// ---- POUs/_Exclude/FB_PACK_WriteOCVFileLoop_v3.TcPOU
(* scan and validate Outers, generate OAC file for new valid Outers *)
FUNCTION_BLOCK FB_PACK_WriteOCVFileLoop_v3
VAR_INPUT
	bExecute						: BOOL;			(* scan for completed Outer *)
	ePackAggregationMode			: E_SYSTEM_PackAggregationMode ;
	strLocalOCVPath				: STRING(50);	(* OCV folder path *)
	nPacksPerOuter				: INT;
	nPackPos1						: INT 	:=1;
	nPackPos2						: INT	:=2;
	nOCVControlCheckStatus		: BYTE;
	aDisablePackAggregCamera	: ARRAY[1..3] OF BOOL;
	stDuplicatedItem				: ST_RejectItems;(*stPackRejectReasons.stPackCodesDuplicated*)
	stCTDateTime					: ST_SYSTEM_DateTime;
END_VAR
VAR_IN_OUT
	stCodeInfo_Pack				: ST_CodeInfo;
	stCodeInfo_Intermediate		: ST_CodeInfo;
	(*aInterimCodeQueue			: ARRAY[1..cMAX_INTERMEDIATE_CODE_QUEUE] OF T_MaxString;*)
	aOCVPackStatus				: ARRAY[1..cMAX_OUTER_STATUS_QUEUE] OF ST_OUTER_Status;	(* Outer status array *)
	stMetsEfficiency				: ST_NOVRAM_METS_Inspection;
	stShiftItemProduced			: ST_KPI_ItemsProduced;
	stProdItemProduced			: ST_KPI_ItemsProduced;
	stLastOCVStatus				: ST_OUTER_Status;	(* Outer status *)
END_VAR
VAR_OUTPUT
	bDone							: BOOL;			(* TRUE = validation complete *)
	bBusy							: BOOL;			(* TRUE = validation in progress *)
	bError							: BOOL;			(* TRUE = validation error *)
	nErrorID						: UDINT;			(* error ID *)
	sOCVFile1						: T_OCV_Filename;	(* OCV file name *)
	sOCVFile2						: T_OCV_Filename;	(* OCV file name *)
	sDeletedOCVFile1				: T_OCV_Filename;
	sDeletedOCVFile2				: T_OCV_Filename;
	bPackCodeDuplicate			: BOOL;
	bInterimCodeDuplicate		: BOOL;
	nWriteOCVError				: UINT;
	nLastTriggerID					: UDINT;
	nOCVFilesCreated				: UDINT;			(* OCV files created *)
	nOCVFilesDeleted				: UINT;
	nOutersStoredInOCV			: UDINT;
	nLinkedPackInOCV				: UDINT;
	nWriteErrorCounter			: UINT;
	bOCVUpdated					: BOOL;
	bOCVValidated					: BOOL;
	stLastValidatedOCV			: ST_OUTER_Status;	(* Outer status *)
	sPackCodesResultToOCV		: T_LongSTRING;
END_VAR
VAR
	fbExecute					: R_TRIG;
	tonTimeOut				: TON;
	rtTimeOutExec				: R_TRIG;
	eState						: E_OCV_State;
	eErrorState					: E_OCV_State;
	eCodeAIType				: E_CodeAIType;
	nMaxOuterIndex			: INT;
	nOuterIndex				: INT;
	nSourceIndex				: INT;
	nPackIndex				: INT;

	bUseIntermediateCode		: BOOL;
	stOCVStatus				: ST_OUTER_Status;	(* Outer status *)

(******************************************************************************)

	fbChekcDupPackCode			: FB_PACK_DuplicatesPackCodes;
	fbPackInspectionEfficency		: FB_KPI_PackEfficiency;
	fbValidateOCVContent			: FB_PACK_ValidateOCVContent;

	aAggregationCodesValid			: ARRAY[1..2] OF  BOOL;
	aDeleteOCVCodesValid			: ARRAY[1..2] OF BOOL;
(******************************************************************************)

	fbWriteOCVFile				: FB_OCV_WriteFile;
	(*sOCVFileName				: T_MaxString;*)
	fbMoveOCVFile			: FB_FILE_Move;

	nOCVLogIndex		: UINT;
	sLocalTargetPath	: STRING(255);

END_VAR


(* monitor rising edge of bExecute *)
fbExecute(CLK := bExecute);

(* monitor Busy timeout *)
tonTimeOut(
	IN:=nSourceIndex <> 0,
	 PT:=cONE_SECOND,
	Q=>
);

rtTimeOutExec(CLK:= tonTimeOut.Q);

IF rtTimeOutExec.Q THEN

	bError := TRUE;
	nErrorID := 100;
	IF nSourceIndex > 0 THEN

		aOCVPackStatus[nSourceIndex].sDataSourceTracker 	:= 	'TIMEOUT_S';
		aOCVPackStatus[nSourceIndex].nStatus.7 := TRUE;

		stLastOCVStatus := aOCVPackStatus[nSourceIndex];
		bOCVUpdated	:= TRUE;
		stLastValidatedOCV := aOCVPackStatus[nSourceIndex];
		bOCVValidated	:= TRUE;
	END_IF

	eState := E_OCV_DONE;
END_IF

(* rising edge of bExecute *)
CASE eState OF

	(* idle *)
	E_OCV_IDLE:

		(* scan for completed Outer when OAC files are required *)
		IF fbExecute.Q = TRUE THEN

			(* update outputs *)
			bDone := FALSE;
			bBusy := TRUE;
			bError := FALSE;
			nErrorID := 0;

			(* clear outputs *)
			nOCVFilesCreated := 0;
			nOutersStoredInOCV := 0;
			nLinkedPackInOCV :=0;
			nWriteErrorCounter :=0;

			(*bOCVUpdated	:= FALSE;*)

			(* max Outer index *)
			nMaxOuterIndex := UDINT_TO_INT(SIZEOF(aOCVPackStatus) / SIZEOF(aOCVPackStatus[1]));

			eState := E_OCV_SCAN;

		(* no action required *)
		ELSIF bExecute = FALSE THEN

			(* reset outputs *)
			bDone := FALSE;
			bBusy := FALSE;
			bError := FALSE;
			nErrorID := 0;

		END_IF

	(* scan for completed Outer *)
	E_OCV_SCAN:

		eState := E_OCV_DONE;
		bOCVUpdated	:= FALSE;
		bOCVValidated	:= FALSE;

		(* reset index of Outer to be written to OCV file *)
		nSourceIndex := 0;
		MEMSET(ADR(aAggregationCodesValid), 16#00, SIZEOF(aAggregationCodesValid));
		MEMSET(ADR(aDeleteOCVCodesValid), 16#00, SIZEOF(aDeleteOCVCodesValid));

		bPackCodeDuplicate			:= FALSE;

		 (* scan aOCVPackStatus  backward - ensures that oldest Outer will be written first *)
		FOR nOuterIndex := nMaxOuterIndex TO 1 BY -1 DO
			CASE ePackAggregationMode OF

			E_SYSTEM_PAOL_3CAM:
				(* TriggerID > 0 indicates Outer data present, nStatus = 14 indicates writing data for all 3 cameras, nStatus.6  indicates OCV file has been alread  created, nStatus.7 indicates OCV write error  *)
				IF aOCVPackStatus[nOuterIndex].nTriggerID > 0 AND
					(aOCVPackStatus[nOuterIndex].nStatus.1 OR aDisablePackAggregCamera[1])	AND
					( aOCVPackStatus[nOuterIndex].nStatus.2 OR aDisablePackAggregCamera[2]) 	AND
					( aOCVPackStatus[nOuterIndex].nStatus.3 OR aDisablePackAggregCamera[3]) 	AND
					NOT aOCVPackStatus[nOuterIndex].nStatus.6 		AND
					NOT aOCVPackStatus[nOuterIndex].nStatus.7  		AND
					NOT aOCVPackStatus[nOuterIndex].nStatus.22		AND
					NOT aOCVPackStatus[nOuterIndex].nStatus.23 	THEN

					(* For lightbox system,mapping packcodes to AggregationCodes, used for file name has to be done here, when we are sure if all pack data was plced to OCV record. Those codes will be used to restore OCV data to OAC*)
					AggregationCodes();

					bUseIntermediateCode := FALSE;
					nSourceIndex := nOuterIndex;
					EXIT;
				END_IF

			E_SYSTEM_PAOL_2CAM:
				(* TriggerID > 0 indicates Outer data present, nStatus = 14 indicates writing data for all 3 cameras, nStatus.6  indicates OCV file has been alread  created, nStatus.7 indicates OCV write error  *)
				IF aOCVPackStatus[nOuterIndex].nTriggerID > 0 AND
					(aOCVPackStatus[nOuterIndex].nStatus.1 OR aDisablePackAggregCamera[1])		AND
					( aOCVPackStatus[nOuterIndex].nStatus.2 OR aDisablePackAggregCamera[2]) 	AND
					NOT aOCVPackStatus[nOuterIndex].nStatus.6 		AND
					NOT aOCVPackStatus[nOuterIndex].nStatus.7  		AND
					NOT aOCVPackStatus[nOuterIndex].nStatus.22		AND
					NOT aOCVPackStatus[nOuterIndex].nStatus.23 	THEN

					(* For lightbox system,mapping packcodes to AggregationCodes, used for file name has to be done here, when we are sure if all pack data was plced to OCV record. Those codes will be used to restore OCV data to OAC*)
					AggregationCodes();

					bUseIntermediateCode := FALSE;
					nSourceIndex := nOuterIndex;
					EXIT;
				END_IF

			E_SYSTEM_PLAS_T01:
				(* TriggerID > 0 indicates Outer data present, nStatus = 14 indicates writing data for all 3 cameras, nStatus.6  indicates OCV file has been alread  created, nStatus.7 indicates OCV write error  *)
				(* For linear aggregation system,AggregationCode shuld be already add from temporary coding system camera. This code will be used for file name and to restore OCV data to OAC*)

				IF aOCVPackStatus[nOuterIndex].nTriggerID > 0 		AND
					aOCVPackStatus[nOuterIndex].nStatus.0			AND 	(*OCV Structure rady to store in file *)
					NOT aOCVPackStatus[nOuterIndex].nStatus.6 		AND
					NOT aOCVPackStatus[nOuterIndex].nStatus.7  		AND
					NOT aOCVPackStatus[nOuterIndex].nStatus.22		AND
					NOT aOCVPackStatus[nOuterIndex].nStatus.23 	THEN

					(* For clear wrap system,mapping packcodes to AggregationCodes, used for file name has to be done here, when we are sure if all pack data was plced to OCV record. Those codes will be used to restore OCV data to OAC*)
					(*AggregationCodes();*)

					bUseIntermediateCode := FALSE;
					nSourceIndex := nOuterIndex;
					EXIT;
				END_IF

			E_SYSTEM_PLAS_T02, E_SYSTEM_PLAS_T03, E_SYSTEM_PLAS_T04:
				(* TriggerID > 0 indicates Outer data present, nStatus = 14 indicates writing data for all 3 cameras, nStatus.6  indicates OCV file has been alread  created, nStatus.7 indicates OCV write error  *)
				(* For linear aggregation system,AggregationCode shuld be already add from temporary coding system camera. This code will be used for file name and to restore OCV data to OAC*)

				IF aOCVPackStatus[nOuterIndex].nTriggerID > 0 		AND
					aOCVPackStatus[nOuterIndex].nStatus.0			AND 	(*OCV Structure rady to store in file *)
					NOT aOCVPackStatus[nOuterIndex].nStatus.6 		AND
					NOT aOCVPackStatus[nOuterIndex].nStatus.7  		AND
					NOT aOCVPackStatus[nOuterIndex].nStatus.22		AND
					NOT aOCVPackStatus[nOuterIndex].nStatus.23 	THEN

					(* For NON clear wrap system,mapping packcodes to AggregationCodes form Intrim code, which might be temp stored as barcode for OCV records.
						AggregationCode1 will be used for file name has to be done here, when we are sure if all pack data was plced to OCV record. Those codes will be used to restore OCV data to OAC*)
						(*aOCVPackStatus[nOuterIndex].stOACData.AggregationCodes[1] :=aOCVPackStatus[nOuterIndex].stOACData.Barcode;*) (*solution never tested yet*)

					bUseIntermediateCode := TRUE;
					nSourceIndex := nOuterIndex;
					EXIT;
				END_IF
			END_CASE
		END_FOR

		(* Outer found requiring OAC file to be written *)
		IF nSourceIndex > 0 THEN

			(* copy Outer data from arrOuterStatus *)
			stOCVStatus := aOCVPackStatus[nSourceIndex];

			stMetsEfficiency.OutersProcessing.AtPackAggregCameras := stMetsEfficiency.OutersProcessing.AtPackAggregCameras  + 1;

			eState := E_OCV_VALIDATECONTENT;
		END_IF

	E_OCV_VALIDATECONTENT:

		fbChekcDupPackCode(
			nNumberPackInOuters := nPacksPerOuter,
			sOuterStatus := stOCVStatus,
			stDuplicatedItem := stDuplicatedItem,
			bDuplicateFound =>  bPackCodeDuplicate
			);

		fbPackInspectionEfficency(
			ePackAggregationMode				:= ePackAggregationMode,
			nTotalOutersProcessingByPackAggregCameras	:= stMetsEfficiency.OutersProcessing.AtPackAggregCameras,
			bUseInterimCode						:= bUseIntermediateCode,
			sOuterStatus							:= stOCVStatus,
			aPacksRead							:= stMetsEfficiency.PacksRead,
			aPackPosEfficiency						:= stMetsEfficiency.PackPosEfficiency,
			stPackAggregationEfficiency			:= stMetsEfficiency.PackAggregationEfficiency,
			stMainItemProduced					:= stMetsEfficiency.PackProduced,
			stShiftItemProduced					:= stShiftItemProduced,
			stProdItemProduced					:= stProdItemProduced
			);

		fbValidateOCVContent(
			nOCVControlCheckStatus			:= nOCVControlCheckStatus,
			nPacksPerOuter					:= nPacksPerOuter,
			stCTDateTime						:= stCTDateTime,
			bUseIntermediateCode				:= bUseIntermediateCode,
			stCodeInfo_Pack					:= stCodeInfo_Pack,
			stCodeInfo_Intermediate			:= stCodeInfo_Intermediate,
			(*aInterimCodeQueue				:= aInterimCodeQueue,*)
			stOCVStatus						:= stOCVStatus,
			stNextOCVStatus					:= aOCVPackStatus[nSourceIndex+1],
			bDuplicateInterimFound			=> bInterimCodeDuplicate
			);


		stLastValidatedOCV := stOCVStatus; (*Use for logging data*)
		bOCVValidated	:= TRUE;	(*Use for SFLX solution*)

		IF F_InvalidateASCIIChar(fbValidateOCVContent.aOCVFileCodeName[1]) =	0 	THEN aAggregationCodesValid[1] := nPackPos1 <> 0 OR  bUseIntermediateCode;  	END_IF
		IF F_InvalidateASCIIChar(fbValidateOCVContent.aOCVFileCodeName[2]) =	0 	THEN aAggregationCodesValid[2] := nPackPos2 <> 0; 		END_IF

		IF (aAggregationCodesValid[1] OR aAggregationCodesValid[2]) THEN
			eState := E_OCV_WRITEDATA;
		ELSE

			stOCVStatus.nStatus.7 := TRUE;

			IF fbValidateOCVContent.bDuplicatePackFound THEN
				eState := E_OCV_MOVEFILE1;
			ELSE
				eState := E_OCV_UPDATESTATUS;
			END_IF

			nWriteErrorCounter := nWriteErrorCounter+1;
		END_IF

	(* write OCVC file *)
	E_OCV_WRITEDATA:

		IF fbValidateOCVContent.bEmptyAggregationCode 		THEN

			sLocalTargetPath := CONCAT(strLocalOCVPath,'Empty\');

		ELSIF fbValidateOCVContent.bInvalidPackFound 			OR
				fbValidateOCVContent.bDuplicatePackFound 		OR
				fbValidateOCVContent.bDuplicateInterimFound 	THEN

			sLocalTargetPath := CONCAT(strLocalOCVPath,'Error\');
		ELSE
			sLocalTargetPath := strLocalOCVPath;
		END_IF

		(* write OCV file *)
		fbWriteOCVFile(
			bExecute					:= TRUE,
			sTargetPath				:= sLocalTargetPath,
			ePackAggregationMode	:= ePackAggregationMode,
			nPacksPerOuter			:= nPacksPerOuter,
			aOCVFileCodeName		:= fbValidateOCVContent.aOCVFileCodeName,  (*strAggregationCodes is a table*)
			bSkipWriteFile1			:= NOT aAggregationCodesValid[1],
			bSkipWriteFile2			:= NOT aAggregationCodesValid[2],
			stOCVPackStatus			:= stOCVStatus
			);
		(* write OCV file complete *)
		IF fbWriteOCVFile.bDone  THEN

			sOCVFile1 := fbWriteOCVFile.sOCVFile1;
			sOCVFile2 := fbWriteOCVFile.sOCVFile2;

			(* write OCV file completed OK *)
			IF NOT  fbWriteOCVFile.bError THEN

				(* count OCV files written *)
				nOCVFilesCreated := nOCVFilesCreated + fbWriteOCVFile.nStoredFiles;
				nOutersStoredInOCV := nOutersStoredInOCV + 1;

				nLastTriggerID :=  stOCVStatus.nTriggerID;

				(* update stOCVStatus - OCV file written OK *)
				stOCVStatus.nStatus.6 := TRUE;
			ELSE
				bError := TRUE;
				nErrorID := fbWriteOCVFile.nErrorID + 1000;

				(* update stOCVStatus - OCV file write error  - general error for OCV *)
				nWriteOCVerror := nWriteOCVerror +1;
				stOCVStatus.nStatus.7 := TRUE;
				eErrorState := eState;
			END_IF

			IF fbValidateOCVContent.bDuplicatePackFound  THEN
				eState := E_OCV_MOVEFILE1;
			ELSE
				eState := E_OCV_UPDATESTATUS;
			END_IF
			(* close off fbWriteOCVFile*)
			fbWriteOCVFile(bExecute := FALSE);
		END_IF

	(* delete OCV to error folder *)
	E_OCV_MOVEFILE1:

		IF F_InvalidateASCIIChar(fbValidateOCVContent.aOCVFileCodeToDelete[1]) = 0 	THEN aDeleteOCVCodesValid[1] := nPackPos1 <> 0 OR  bUseIntermediateCode;  	END_IF

		(*sOCVFileName := F_CONCAT3('OCV_', fbValidateOCVContent.aOCVFileCodeToDelete[1], '.xml');*)
		(* delete OCV file *)
		fbMoveOCVFile(
				bExecute			:= aDeleteOCVCodesValid[1],
				strPathSource		:= strLocalOCVPath,
				strPathTarget		:= CONCAT(strLocalOCVPath,'Error\' ),
				strFileName		:= fbValidateOCVContent.aOCVFileCodeToDelete[1],
				tTimeout			:= cHALF_SECOND
		);

		(* delete file complete *)
		IF NOT fbMoveOCVFile.bBusy  OR NOT aDeleteOCVCodesValid[1] THEN

			(* delete  file completed OK *)
			IF NOT  fbMoveOCVFile.bError THEN

				(* update counter *)
				IF  aDeleteOCVCodesValid[1] THEN
					nOCVFilesDeleted := nOCVFilesDeleted + 1;
					sDeletedOCVFile1 := fbMoveOCVFile.strLastFileMoved;
				END_IF
			(* delete command error or file not found *)
			ELSE

				bError := TRUE;
				nErrorID := fbMoveOCVFile.nErrorID + 2000;
				eErrorState := eState;
			END_IF

			(* close off fbDeleteOCVFile *)
			fbMoveOCVFile(bExecute := FALSE);

			eState := E_OCV_MOVEFILE2;
		END_IF

	(* delete OCV to error folder *)
	E_OCV_MOVEFILE2:

		IF F_InvalidateASCIIChar(fbValidateOCVContent.aOCVFileCodeToDelete[2]) = 0 	THEN aDeleteOCVCodesValid[2] := nPackPos2 <> 0; 		END_IF

		(*sOCVFileName := F_CONCAT3('OCV_', fbValidateOCVContent.aOCVFileCodeToDelete[2], '.xml');*)
		(* delete OCV file *)
		fbMoveOCVFile(
				bExecute			:= aDeleteOCVCodesValid[2],
				strPathSource		:= strLocalOCVPath,
				strPathTarget		:= CONCAT(strLocalOCVPath,'Error\' ),
				strFileName		:= fbValidateOCVContent.aOCVFileCodeToDelete[2],
				tTimeout			:= cHALF_SECOND
		);

		(* delete file complete *)
		IF NOT fbMoveOCVFile.bBusy  OR NOT aDeleteOCVCodesValid[2] THEN

			(* delete  file completed OK *)
			IF NOT  fbMoveOCVFile.bError  THEN

				(* update counter *)
				IF aDeleteOCVCodesValid[2] THEN
					nOCVFilesDeleted := nOCVFilesDeleted + 1;
					sDeletedOCVFile2 := fbMoveOCVFile.strLastFileMoved;
				END_IF
			(* delete command error or file not found *)
			ELSE

				bError := TRUE;
				nErrorID := fbMoveOCVFile.nErrorID + 3000;
				eErrorState := eState;
			END_IF
			(* close off fbDeleteOCVFile *)
			fbMoveOCVFile(bExecute := FALSE);

			eState := E_OCV_UPDATESTATUS;
		END_IF

	(* update Outer status *)
	E_OCV_UPDATESTATUS:

		nSourceIndex := 0;
		(* move stOCVStatus data back to shift reg *)
		FOR nOuterIndex := 1 TO nMaxOuterIndex DO

			(* matching nTriggerID found *)
			IF aOCVPackStatus[nOuterIndex].nTriggerID = stOCVStatus.nTriggerID THEN

				(* move updated Outer data to shift reg *)
				aOCVPackStatus[nOuterIndex] := stOCVStatus;
				stLastOCVStatus := stOCVStatus;

				nLinkedPackInOCV :=nLinkedPackInOCV + stOCVStatus.stOACData.NumberOfLinkedPacks;
				bOCVUpdated	:= TRUE;

				sPackCodesResultToOCV	:= '';
				sPackCodesResultToOCV := F_CONCAT5('[', RIGHT(stLastOCVStatus.stOACData.AggregationCodes[1],7),']:[',RIGHT(stLastOCVStatus.stOACData.AggregationCodes[2],7),']');
				FOR nOCVLogIndex := 1 TO MIN(nPacksPerOuter ,cMAX_PACKS_PER_OUTER) BY 1 DO
					sPackCodesResultToOCV :=F_LongCONCAT(sPackCodesResultToOCV, '     ');
					sPackCodesResultToOCV := F_LongCONCAT(sPackCodesResultToOCV, RIGHT(F_CODE_GetItem(stLastOCVStatus.stOACData.PackCode[nOCVLogIndex], eCodeAIType.SerialCode, stCodeInfo_Pack),7));
				END_FOR

				EXIT;
			END_IF
		END_FOR

		eState := E_OCV_SCAN;

	(* OCV file complete *)
	E_OCV_DONE:

		(* update outputs *)
		bDone := TRUE;
		bBusy := FALSE;

		eState := E_OCV_IDLE;

(* unknown state *)
ELSE

	eState := E_OCV_IDLE;
END_CASE

ACTION AggregationCodes:
IF nPackPos1 <> 0 THEN
	IF aOCVPackStatus[nOuterIndex].aOACPackStatus[nPackPos1] > 1 THEN
		aOCVPackStatus[nOuterIndex].stOACData.AggregationCodes[1] :=aOCVPackStatus[nOuterIndex].stOACData.PackCode[nPackPos1];
	ELSE
		aOCVPackStatus[nOuterIndex].stOACData.AggregationCodes[1] := '';
	END_IF
ELSE
	aOCVPackStatus[nOuterIndex].stOACData.AggregationCodes[1] := '';
END_IF

IF nPackPos2 <> 0 THEN
	IF aOCVPackStatus[nOuterIndex].aOACPackStatus[nPackPos2] > 1 THEN
		aOCVPackStatus[nOuterIndex].stOACData.AggregationCodes[2] :=aOCVPackStatus[nOuterIndex].stOACData.PackCode[nPackPos2];
	ELSE
		aOCVPackStatus[nOuterIndex].stOACData.AggregationCodes[2] := '';
	END_IF
ELSE
	aOCVPackStatus[nOuterIndex].stOACData.AggregationCodes[2] := '';
END_IF
END_ACTION

END_FUNCTION_BLOCK

// ---- POUs/_Exclude/FB_T03_MoveDataToOCVStatus_ORG.TcPOU
FUNCTION_BLOCK FB_T03_MoveDataToOCVStatus_ORG
VAR_INPUT
	bExecute						: BOOL;

	stImageData					: ST_SCANNER_ImageData;	(* image data structure *)
	nExpectedResp					: INT:=1;
	(*nExpectedValidationDepth		: INT;*)
	nPacksPerOuter				: UINT;
	bConfirmOnOuter				: BOOL;
END_VAR
VAR_IN_OUT
	stPackRejectReasons			: ST_RejectReasonsForPack;
	stPackInFeedQueue			: ST_PACK_InfeedQueue; (* Infeed queue *)
	stOCVPackStatus				: ST_OUTER_Status;
	stCodeInfo						: ST_CodeInfo;
END_VAR
VAR_OUTPUT
	bDone							: BOOL;

	nImageDataIndex				: UINT;
	nSearchIndex					: UINT;
	nMoveIndex					: UINT;
	nValidatinIndex				: UINT;

	bOCVStackOutOfSequence		: BOOL;
	bOCVNoConfiramtion			: BOOL;
	bOCVConfirmationNotFound	: BOOL;

	sStackerDataLog				: T_LongSTRING;
END_VAR
VAR
	fbExecute						: R_TRIG;

	nPackIndex					: UINT;
	nLogIndex						: INT;

	nValidationOffset 				: INT;

	aDiagonosticError				: ARRAY[1..10] OF INT;
	aDiagonosticMove				: ARRAY[0..20] OF INT;
END_VAR

VAR CONSTANT
	aPackCodeMapping2x5		: ARRAY[1..cMAX_PACKS_PER_OUTER] OF INT :=[ 	9, 8, 7, 6, 5, 4, 3, 2, 1, 0];		(*mapping examples*)
	aPackCodeMapping5x2		: ARRAY[1..cMAX_PACKS_PER_OUTER] OF INT :=[ 	0, 1, 2, 3, 4, 5, 6, 7, 8, 9];		(*mapping examples*)
END_VAR

fbExecute(CLK := bExecute);

IF fbExecute.Q THEN

	bDone := FALSE;
	nMoveIndex	:= 0;
	nSearchIndex 	:=0;		(*initialize in for loop on 1*)
	nImageDataIndex := 0;	(*initialize in for loop on 1*)

	sStackerDataLog	:= '';

	bOCVStackOutOfSequence		:= FALSE;
	bOCVNoConfiramtion			:= FALSE;
	(*bOCVConfirmationNotFound	:= FALSE;*)

	(*nExpectedValidationDepth	:= LIMIT(1, nExpectedValidationDepth, cMAX_CAMERA_PROG_NUMBER);*)

	nValidationOffset :=SEL(bConfirmOnOuter, 0, nExpectedResp);

(*********************************Identify index***************************************************)

	IF stImageData.nCodesRead > 0 THEN

		FOR nImageDataIndex := 1 TO stImageData.nCodesRead DO
			FOR nSearchIndex :=1 TO cMAX_PACK_INFEED_QUEUE DO

				IF stImageData.aCodeData[nImageDataIndex].strDataString  = stPackInFeedQueue.aPackQueue[nSearchIndex].sPackCode AND
					stPackInFeedQueue.aPackQueue[nSearchIndex].sPackCode <> '' THEN

					IF nSearchIndex > stImageData.aCodeData[nImageDataIndex].nProgramNo THEN
						nMoveIndex := nSearchIndex-stImageData.aCodeData[nImageDataIndex].nProgramNo +nValidationOffset;  (*add nExpectedResp as an option*)
						EXIT;
					END_IF
				END_IF
			END_FOR

			IF nMoveIndex > 0 THEN
				EXIT;
			END_IF
		END_FOR

	ELSIF stImageData.nCodesRead = 0 AND stPackInFeedQueue.nIndex = nPacksPerOuter THEN
		
		nMoveIndex := stPackInFeedQueue.nIndex;
	END_IF

sStackerDataLog	:= F_CONCAT3('MOVED ITEM [', UINT_TO_STRING(nMoveIndex), ']:');

(*********************************Validation***************************************************)

	IF	bOCVConfirmationNotFound AND nMoveIndex <> 0 THEN		(*reject next outer after one with read code bou confirmation not found*)

		sStackerDataLog	:= CONCAT(sStackerDataLog, '[X]');

		aDiagonosticError[1]	:=  aDiagonosticError[1] + 1;
		bOCVConfirmationNotFound := FALSE;
		bOCVStackOutOfSequence := TRUE;

	ELSIF	stImageData.nCodesRead = 0 AND nMoveIndex = nPacksPerOuter THEN		(*move without confirmation found - temp blocked*)

		aDiagonosticError[2]	:=  aDiagonosticError[2] + 1;
		bOCVNoConfiramtion := TRUE;

	ELSIF nMoveIndex = 0 AND stImageData.nCodesRead <> 0 THEN			(*Confirmation code read but not found in infeed*)

		sStackerDataLog	:= CONCAT(sStackerDataLog, '[Y]');

		aDiagonosticError[3]	:=  aDiagonosticError[3] + 1;
		bOCVConfirmationNotFound := TRUE;

	ELSIF nMoveIndex = 0 THEN		(*Confirmation code not found becouse camera not read*)

		sStackerDataLog	:= CONCAT(sStackerDataLog, '[Z]');

		aDiagonosticError[4]	:=  aDiagonosticError[4] + 1;
		bOCVConfirmationNotFound := TRUE;

	ELSIF  stImageData.nCodesRead <> nExpectedResp (*nExpectedValidationDepth*) THEN	(*no read or not enough code read found but at leas one code read and found*)

		aDiagonosticError[5]	:=  aDiagonosticError[5] + 1;
		bOCVStackOutOfSequence := TRUE;

	ELSIF nMoveIndex > nPacksPerOuter THEN		(*f.ex phisical packs remode form line*)

		aDiagonosticError[6]	:=  aDiagonosticError[6] + 1;
		bOCVStackOutOfSequence := TRUE;

	ELSIF nMoveIndex < nPacksPerOuter THEN		(*f.ex phantom packs passed form the line or queue was deleted*)

		aDiagonosticError[7]	:=  aDiagonosticError[7] + 1;
		bOCVStackOutOfSequence := TRUE;

		IF nMoveIndex < 20 THEN	aDiagonosticMove[nMoveIndex] :=  aDiagonosticMove[nMoveIndex] + 1; END_IF

		aDiagonosticError[8]	:=  aDiagonosticError[8] + 1;
		bOCVStackOutOfSequence := TRUE;

	ELSIF nMoveIndex = nPacksPerOuter  AND
			stImageData.nCodesRead > 0	AND
			nMoveIndex  <= cMAX_PACK_INFEED_QUEUE - cMAX_CAMERA_PROG_NUMBER	THEN

		(*Check all reaming codes in the comfirmation stack*)
		FOR nValidatinIndex := 1 TO stImageData.nCodesRead DO														(*nMovePsotion - nExpectedResp as an option*)
			IF stImageData.aCodeData[nValidatinIndex].strDataString <> stPackInFeedQueue.aPackQueue[nMoveIndex + stImageData.aCodeData[nValidatinIndex].nProgramNo - nValidationOffset].sPackCode(* AND
				stPackInFeedQueue.aPackQueue[nMoveIndex + stImageData.aCodeData[nValidatinIndex].nProgramNo - nValidationOffset].sPackCode <> ''*)  THEN (*More restricted to reject if comapre with empty*)

				aDiagonosticError[9]	:=  aDiagonosticError[9] + 1;
				bOCVStackOutOfSequence := TRUE;
				EXIT;
			END_IF
		END_FOR
	ELSE
		aDiagonosticError[10]	:=  aDiagonosticError[10] + 1;
		bOCVStackOutOfSequence := TRUE;
	END_IF

(*********************************Fill up OCV pack data***************************************************)

	IF NOT bOCVStackOutOfSequence 		AND
		NOT bOCVNoConfiramtion 			AND
		NOT bOCVConfirmationNotFound  	THEN		(*temp for now included bOCVNoConfiramtion*)

		FOR nPackIndex := 1 TO LIMIT(1, nPacksPerOuter, cMAX_PACKS_PER_OUTER) DO

			(* to avoid incorect mapping in PackCodeMapping declaration, where array index <0 *)
			IF nMoveIndex >  aPackCodeMapping2x5[nPackIndex] AND nPacksPerOuter > 0 THEN
				stOCVPackStatus.stOACData.PackCode[nPackIndex] := stPackInFeedQueue.aPackQueue[nMoveIndex - aPackCodeMapping2x5[nPackIndex]].sPackCode;
				stOCVPackStatus.aPackCodeFilledIn[nPackIndex] := stPackInFeedQueue.aPackQueue[nMoveIndex -aPackCodeMapping2x5[nPackIndex]].ePackCodeFilledIn;
				stOCVPackStatus.aPackCodes[nPackIndex].sBuffer[1].strCode := stPackInFeedQueue.aPackQueue[nMoveIndex -aPackCodeMapping2x5[nPackIndex]].stPackCodeData.strDataString;

				stOCVPackStatus.aOACPackStatus[nPackIndex]	:= stPackInFeedQueue.aPackQueue[nMoveIndex -aPackCodeMapping2x5[nPackIndex]].nPackStatus;
				stOCVPackStatus.stOACData.PackRejectID[nPackIndex] :=  stPackInFeedQueue.aPackQueue[nMoveIndex -aPackCodeMapping2x5[nPackIndex]].nPackRejectID;
				stOCVPackStatus.stOACData.PackRejectCode[nPackIndex] := stPackInFeedQueue.aPackQueue[nMoveIndex -aPackCodeMapping2x5[nPackIndex]].sPackRejectCode;
			ELSE
				EXIT;  	(*stOCVPackStatus remain empty - wrong input parameters*)
			END_IF
		END_FOR
	ELSE

		FOR nPackIndex := 1 TO LIMIT(1, nPacksPerOuter, cMAX_PACKS_PER_OUTER) DO

			IF nPacksPerOuter > 0 THEN
				stOCVPackStatus.stOACData.PackCode[nPackIndex] :=  cCODE_OVERWIRTTEN;
				stOCVPackStatus.aPackCodeFilledIn[nPackIndex] := E_PACK_CODEOVERWRITTEN;
				stOCVPackStatus.aPackCodes[nPackIndex].sBuffer[1].strCode :=  cCODE_OVERWIRTTEN;
		
				stOCVPackStatus.aOACPackStatus[nPackIndex]	:= 1;
				stOCVPackStatus.stOACData.PackRejectID[nPackIndex] :=  stPackRejectReasons.stPackCodesOverwritten.nRejectID;
				stOCVPackStatus.stOACData.PackRejectCode[nPackIndex] := stPackRejectReasons.stPackCodesOverwritten.sMetsDisplayCode;
			ELSE
				EXIT;	(*stOCVPackStatus remain empty - wrong input parameters*)
			END_IF
		END_FOR
	END_IF

(*********************************Log Move Pack Infeed Queue***************************************************)

	IF nMoveIndex <> 0 THEN
		FOR nLogIndex :=1 TO nMoveIndex  DO
			sStackerDataLog :=F_LongCONCAT(sStackerDataLog, '   ');
			sStackerDataLog :=F_LongCONCAT(sStackerDataLog, RIGHT(F_CODE_GetItem(stPackInFeedQueue.aPackQueue[nLogIndex].sPackCode, eCodeAIType.SerialCode, stCodeInfo), 5));
		END_FOR
	END_IF

(*********************************Move Pack Infeed Queue***************************************************)

	IF nMoveIndex <> 0 THEN
		(* move remaining Outers forward in sInfeedQueue and update index pointer *)
		IF cMAX_PACK_INFEED_QUEUE  > nMoveIndex  THEN
	
			MEMMOVE(ADR(stPackInFeedQueue.aPackQueue[1]), ADR(stPackInFeedQueue.aPackQueue[nMoveIndex + 1]),
											 (cMAX_PACK_INFEED_QUEUE- nMoveIndex) * SIZEOF(stPackInFeedQueue.aPackQueue[1]));
			stPackInFeedQueue.nIndex := LIMIT(0, stPackInFeedQueue.nIndex - nMoveIndex,cMAX_PACK_INFEED_QUEUE);
	
		END_IF
	
		(* clear all data for empty Packs in PackInFeedQueue -> from Index + 1 till end of queue *)
		IF cMAX_PACK_INFEED_QUEUE > stPackInFeedQueue.nIndex  THEN

			MEMSET(ADR(stPackInFeedQueue.aPackQueue[stPackInFeedQueue.nIndex + 1]), 16#00,
											(cMAX_PACK_INFEED_QUEUE - stPackInFeedQueue.nIndex ) * SIZEOF(stPackInFeedQueue.aPackQueue[1]));
		END_IF
	END_IF
(****************************************************************************************************************************************************************)

	bDone := TRUE;
ELSE
	bDone := FALSE;

END_IF

END_FUNCTION_BLOCK

// ---- POUs/_Exclude/FSS2/FB_FSS2_BuildXMLData.TcPOU
FUNCTION_BLOCK FB_FSS2_BuildXMLData
VAR_INPUT
	bExecute		: BOOL;
	nCartonsPerMasterCase	:UINT	:=50;
END_VAR
VAR_IN_OUT
	stAgregationData	 			: ST_CHM_Data;		(* case data to be written to XML *)
END_VAR
VAR_OUTPUT
	bDone			: BOOL;
	nImageByte		: INT;		(* total bytes for OAC template *)
	arrXMLImage		: ARRAY[0..4096] OF BYTE;
END_VAR
VAR
	fbExecute		: R_TRIG;
	nOuterIndex		: INT;		(* Outer index when building for CAC file *)

	strString		: STRING(255);
	(*nStringLen		: INT;*)

END_VAR

(* rising edge of bExecute *)
fbExecute(CLK := bExecute);

(* rising edge of bExecute *)
IF fbExecute.Q = TRUE THEN

	(* update outputs *)
	bDone := FALSE;

	(* clear output array and reset byte counter *)
	MEMSET(ADR(arrXMLImage), 16#00, SIZEOF(arrXMLImage));
	nImageByte := 0;


(********************XML FILE BIULD SEQTION****************************)
(* XML file version *)
strString := '<?xml version="1.0" encoding="utf-8"?>$R$N';
MEMMOVE(ADR(arrXMLImage[nImageByte]), ADR(strString), LEN(strString));
nImageByte := nImageByte + LEN(strString);

(* XPath leading tag *)
strString := '<GenericHierarchyList xmlns:xsi="http://www.w3.org/2001/XMLSchema-instance" xsi:noNamespaceSchemaLocation="TNTGenericHierarchy.xsd"> $R$N';
MEMMOVE(ADR(arrXMLImage[nImageByte]), ADR(strString), LEN(strString));
nImageByte := nImageByte + LEN(strString);

	(* RequestID *)
	strString := F_CONCAT3('$T<RequestID>','' , '</RequestID>$R$N');
	MEMMOVE(ADR(arrXMLImage[nImageByte]), ADR(strString), LEN(strString));
	nImageByte := nImageByte + LEN(strString);

	(* Sender *)
	strString := F_CONCAT3('$T<Sender>', 'TNTLS' , '</Sender>$R$N');
	MEMMOVE(ADR(arrXMLImage[nImageByte]), ADR(strString), LEN(strString));
	nImageByte := nImageByte + LEN(strString);

	(* GenericHierarchy *)
	strString := '$T<GenericHierarchy>$R$N';
	MEMMOVE(ADR(arrXMLImage[nImageByte]), ADR(strString), LEN(strString));
	nImageByte := nImageByte + LEN(strString);

		(* User *)
		strString := F_CONCAT3('$T$T<User>','TNTLS', '</User>$R$N');
		MEMMOVE(ADR(arrXMLImage[nImageByte]), ADR(strString), LEN(strString));
		nImageByte := nImageByte + LEN(strString);

		(* Timestamp *)
		strString := F_CONCAT3('$T$T<Timestamp>', stAgregationData.MessageHeader.CreationTimeLocalUTC, '</Timestamp>$R$N');
		MEMMOVE(ADR(arrXMLImage[nImageByte]), ADR(strString), LEN(strString));
		nImageByte := nImageByte + LEN(strString);

		(* PackLevel *)
		strString := F_CONCAT3('$T$T<PackLevel>','MASTERCASE', '</PackLevel>$R$N');
		MEMMOVE(ADR(arrXMLImage[nImageByte]), ADR(strString), LEN(strString));
		nImageByte := nImageByte + LEN(strString);

		(* Parent *)
		strString := '$T$T<Parent>$R$N';
		MEMMOVE(ADR(arrXMLImage[nImageByte]), ADR(strString), LEN(strString));
		nImageByte := nImageByte + LEN(strString);
	
			(* ID *)
			strString := F_CONCAT3('$T$T$T<ID>',stAgregationData.GenericHierarchy.CaseItem.Identity.ID, '</ID>$R$N');
			MEMMOVE(ADR(arrXMLImage[nImageByte]), ADR(strString), LEN(strString));
			nImageByte := nImageByte + LEN(strString);
	
			(* GTIN *)
			strString := F_CONCAT3('$T$T$T<GTIN>', stAgregationData.GenericHierarchy.CaseItem.Identity.GTIN, '</GTIN>$R$N');
			MEMMOVE(ADR(arrXMLImage[nImageByte]), ADR(strString), LEN(strString));
			nImageByte := nImageByte + LEN(strString);

		(*/Parent *)
		strString := '$T$T</Parent>$R$N';
		MEMMOVE(ADR(arrXMLImage[nImageByte]), ADR(strString), LEN(strString));
		nImageByte := nImageByte + LEN(strString);

		(*Childs *)
		strString := '$T$T<Childs>$R$N';
		MEMMOVE(ADR(arrXMLImage[nImageByte]), ADR(strString), LEN(strString));
		nImageByte := nImageByte + LEN(strString);

			(* ChildDefaults *)
			strString := '$T$T$T<ChildDefaults>$R$N';
			MEMMOVE(ADR(arrXMLImage[nImageByte]), ADR(strString), LEN(strString));
			nImageByte := nImageByte + LEN(strString);
		
				(* ProductNo *)
				strString := F_CONCAT3('$T$T$T$T<ProductNo>',stAgregationData.GenericHierarchy.CaseItem.Content.DefaultIdentity.SKU, '</ProductNo>$R$N');
				MEMMOVE(ADR(arrXMLImage[nImageByte]), ADR(strString), LEN(strString));
				nImageByte := nImageByte + LEN(strString);
		
				(* GTIN *)
				strString := F_CONCAT3('$T$T$T$T<GTIN>', stAgregationData.GenericHierarchy.CaseItem.Content.DefaultIdentity.GTIN, '</GTIN>$R$N');
				MEMMOVE(ADR(arrXMLImage[nImageByte]), ADR(strString), LEN(strString));
				nImageByte := nImageByte + LEN(strString);
	
			(*/ChildDefaults *)
			strString := '$T$T$T</ChildDefaults>$R$N';
			MEMMOVE(ADR(arrXMLImage[nImageByte]), ADR(strString), LEN(strString));
			nImageByte := nImageByte + LEN(strString);

		(* for each case Child*)
		FOR nOuterIndex := 1 TO nCartonsPerMasterCase DO

			(* <Child  index="xx"> field *)
			strString := '$T$T$T<Child>$R$N';
			MEMMOVE(ADR(arrXMLImage[nImageByte]), ADR(strString), LEN(strString));
			nImageByte := nImageByte + LEN(strString);
		
				(* ID *)
				strString := F_CONCAT3('$T$T$T$T<ID>',stAgregationData.GenericHierarchy.CaseItem.Content.arrOuterItem[nOuterIndex].Identity.ID, '</ID>$R$N');
				MEMMOVE(ADR(arrXMLImage[nImageByte]), ADR(strString), LEN(strString));
				nImageByte := nImageByte + LEN(strString);

			(*/Child *)
			strString := '$T$T$T</Child>$R$N';
			MEMMOVE(ADR(arrXMLImage[nImageByte]), ADR(strString), LEN(strString));
			nImageByte := nImageByte + LEN(strString);

		END_FOR

		(*/Childs *)
		strString := '$T$T</Childs>$R$N';
		MEMMOVE(ADR(arrXMLImage[nImageByte]), ADR(strString), LEN(strString));
		nImageByte := nImageByte + LEN(strString);

		(* Location *)
		strString := '$T$T<Location>$R$N';
		MEMMOVE(ADR(arrXMLImage[nImageByte]), ADR(strString), LEN(strString));
		nImageByte := nImageByte + LEN(strString);
	
			(* ID *)
			strString := F_CONCAT3('$T$T$T<ID>',stAgregationData.GenericHierarchy.CaseItem.Content.DefaultIdentity.ProductionLine, '</ID>$R$N');
			MEMMOVE(ADR(arrXMLImage[nImageByte]), ADR(strString), LEN(strString));
			nImageByte := nImageByte + LEN(strString);

		(*/Location *)
		strString := '$T$T</Location>$R$N';
		MEMMOVE(ADR(arrXMLImage[nImageByte]), ADR(strString), LEN(strString));
		nImageByte := nImageByte + LEN(strString);

		(* CartonsPerMasterCase *)
		strString := F_CONCAT3('$T$T<CartonsPerMasterCase>',stAgregationData.GenericHierarchy.CaseItem.Content.ExpectedItemCount, '</CartonsPerMasterCase>$R$N');
		MEMMOVE(ADR(arrXMLImage[nImageByte]), ADR(strString), LEN(strString));
		nImageByte := nImageByte + LEN(strString);

	(* /GenericHierarchy *)
	strString := '$T</GenericHierarchy>$R$N';
	MEMMOVE(ADR(arrXMLImage[nImageByte]), ADR(strString), LEN(strString));
	nImageByte := nImageByte + LEN(strString);

(* /GenericHierarchyList *)
strString := '$T</GenericHierarchyList>$R$N';
MEMMOVE(ADR(arrXMLImage[nImageByte]), ADR(strString), LEN(strString));
nImageByte := nImageByte + LEN(strString);

(*****************************************************************************)


	(* update outputs *)
	bDone := TRUE;

(* unknown state *)
ELSIF bExecute = FALSE THEN

	(* clear outputs *)
	bDone := FALSE;
END_IF

END_FUNCTION_BLOCK

// ---- POUs/_Exclude/FSS2/FB_FSS2_BuildXMLDataForGMES.TcPOU
FUNCTION_BLOCK FB_FSS2_BuildXMLDataForGMES
VAR_INPUT
	bExecute		: BOOL;
	nCartonsPerMasterCase	:UINT	:=50;
END_VAR
VAR_IN_OUT
	stAgregationData	 			: ST_CHM_Data;		(* case data to be written to XML *)
END_VAR
VAR_OUTPUT
	bDone			: BOOL;
	nImageByte		: INT;		(* total bytes for OAC template *)
	arrXMLImage		: ARRAY[0..2048] OF BYTE;
END_VAR
VAR
	fbExecute		: R_TRIG;

	strString		: STRING(255);
	(*nStringLen		: INT;*)

END_VAR

(* rising edge of bExecute *)
fbExecute(CLK := bExecute);

(* rising edge of bExecute *)
IF fbExecute.Q = TRUE THEN

	(* update outputs *)
	bDone := FALSE;

	(* clear output array and reset byte counter *)
	MEMSET(ADR(arrXMLImage), 16#00, SIZEOF(arrXMLImage));
	nImageByte := 0;


(********************XML FILE BIULD SEQTION****************************)
(* XML file version *)
strString := '<?xml version="1.0" encoding="utf-8"?>$R$N';
MEMMOVE(ADR(arrXMLImage[nImageByte]), ADR(strString), LEN(strString));
nImageByte := nImageByte + LEN(strString);

(* XPath leading tag *)
strString := '<GenericHierarchyList xsi:noNamespaceSchemaLocation="TNTGenericHierarchy.xsd" xmlns:xsi="http://www.w3.org/2001/XMLSchema-instance"> $R$N';
MEMMOVE(ADR(arrXMLImage[nImageByte]), ADR(strString), LEN(strString));
nImageByte := nImageByte + LEN(strString);

	(* RequestID *)
	strString := F_CONCAT3('$T<RequestID>','' , '</RequestID>$R$N');
	MEMMOVE(ADR(arrXMLImage[nImageByte]), ADR(strString), LEN(strString));
	nImageByte := nImageByte + LEN(strString);

	(* Sender *)
	strString := F_CONCAT3('$T<Sender>', 'TNTLS' , '</Sender>$R$N');
	MEMMOVE(ADR(arrXMLImage[nImageByte]), ADR(strString), LEN(strString));
	nImageByte := nImageByte + LEN(strString);

	(* GenericHierarchy *)
	strString := '$T<GenericHierarchy>$R$N';
	MEMMOVE(ADR(arrXMLImage[nImageByte]), ADR(strString), LEN(strString));
	nImageByte := nImageByte + LEN(strString);

		(* User *)
		strString := F_CONCAT3('$T$T<User>','TNTLS', '</User>$R$N');
		MEMMOVE(ADR(arrXMLImage[nImageByte]), ADR(strString), LEN(strString));
		nImageByte := nImageByte + LEN(strString);

		(* Timestamp *)
		strString := F_CONCAT3('$T$T<Timestamp>', stAgregationData.MessageHeader.CreationTimeLocalUTC, '</Timestamp>$R$N');
		MEMMOVE(ADR(arrXMLImage[nImageByte]), ADR(strString), LEN(strString));
		nImageByte := nImageByte + LEN(strString);

		(* PackLevel *)
		strString := F_CONCAT3('$T$T<PackLevel>','MASTERCASE', '</PackLevel>$R$N');
		MEMMOVE(ADR(arrXMLImage[nImageByte]), ADR(strString), LEN(strString));
		nImageByte := nImageByte + LEN(strString);

		(* Parent *)
		strString := '$T$T<Parent>$R$N';
		MEMMOVE(ADR(arrXMLImage[nImageByte]), ADR(strString), LEN(strString));
		nImageByte := nImageByte + LEN(strString);
	
			(* ID *)
			strString := F_CONCAT3('$T$T$T<ID>',stAgregationData.GenericHierarchy.CaseItem.Identity.ID, '</ID>$R$N');
			MEMMOVE(ADR(arrXMLImage[nImageByte]), ADR(strString), LEN(strString));
			nImageByte := nImageByte + LEN(strString);
	
			(* GTIN *)
			strString := F_CONCAT3('$T$T$T<GTIN>', stAgregationData.GenericHierarchy.CaseItem.Identity.GTIN, '</GTIN>$R$N');
			MEMMOVE(ADR(arrXMLImage[nImageByte]), ADR(strString), LEN(strString));
			nImageByte := nImageByte + LEN(strString);

		(*/Parent *)
		strString := '$T$T</Parent>$R$N';
		MEMMOVE(ADR(arrXMLImage[nImageByte]), ADR(strString), LEN(strString));
		nImageByte := nImageByte + LEN(strString);

		(*Childs *)
		strString := '$T$T<Childs>$R$N';
		MEMMOVE(ADR(arrXMLImage[nImageByte]), ADR(strString), LEN(strString));
		nImageByte := nImageByte + LEN(strString);

			(* ChildDefaults *)
			strString := '$T$T$T<ChildDefaults>$R$N';
			MEMMOVE(ADR(arrXMLImage[nImageByte]), ADR(strString), LEN(strString));
			nImageByte := nImageByte + LEN(strString);
		
				(* ProductNo *)
				strString := F_CONCAT3('$T$T$T$T<ProductNo>',stAgregationData.GenericHierarchy.CaseItem.Content.DefaultIdentity.SKU, '</ProductNo>$R$N');
				MEMMOVE(ADR(arrXMLImage[nImageByte]), ADR(strString), LEN(strString));
				nImageByte := nImageByte + LEN(strString);
		
				(* GTIN *)
				strString := F_CONCAT3('$T$T$T$T<GTIN>', stAgregationData.GenericHierarchy.CaseItem.Content.DefaultIdentity.GTIN, '</GTIN>$R$N');
				MEMMOVE(ADR(arrXMLImage[nImageByte]), ADR(strString), LEN(strString));
				nImageByte := nImageByte + LEN(strString);
	
			(*/ChildDefaults *)
			strString := '$T$T$T</ChildDefaults>$R$N';
			MEMMOVE(ADR(arrXMLImage[nImageByte]), ADR(strString), LEN(strString));
			nImageByte := nImageByte + LEN(strString);

		(*/Childs *)
		strString := '$T$T</Childs>$R$N';
		MEMMOVE(ADR(arrXMLImage[nImageByte]), ADR(strString), LEN(strString));
		nImageByte := nImageByte + LEN(strString);

		(* Location *)
		strString := '$T$T<Location>$R$N';
		MEMMOVE(ADR(arrXMLImage[nImageByte]), ADR(strString), LEN(strString));
		nImageByte := nImageByte + LEN(strString);
	
			(* ID *)
			strString := F_CONCAT3('$T$T$T<ID>',stAgregationData.GenericHierarchy.CaseItem.Content.DefaultIdentity.ProductionLine, '</ID>$R$N');
			MEMMOVE(ADR(arrXMLImage[nImageByte]), ADR(strString), LEN(strString));
			nImageByte := nImageByte + LEN(strString);

		(*/Location *)
		strString := '$T$T</Location>$R$N';
		MEMMOVE(ADR(arrXMLImage[nImageByte]), ADR(strString), LEN(strString));
		nImageByte := nImageByte + LEN(strString);

		(* CartonsPerMasterCase *)
		strString := F_CONCAT3('$T$T<CartonsPerMasterCase>',stAgregationData.GenericHierarchy.CaseItem.Content.ExpectedItemCount, '</CartonsPerMasterCase>$R$N');
		MEMMOVE(ADR(arrXMLImage[nImageByte]), ADR(strString), LEN(strString));
		nImageByte := nImageByte + LEN(strString);

		(* MasterCaseOnly *)
		strString := F_CONCAT3('$T$T<MasterCaseOnly>','false', '</MasterCaseOnly>$R$N');
		MEMMOVE(ADR(arrXMLImage[nImageByte]), ADR(strString), LEN(strString));
		nImageByte := nImageByte + LEN(strString);


	(* /GenericHierarchy *)
	strString := '$T</GenericHierarchy>$R$N';
	MEMMOVE(ADR(arrXMLImage[nImageByte]), ADR(strString), LEN(strString));
	nImageByte := nImageByte + LEN(strString);

(* /GenericHierarchyList *)
strString := '$T</GenericHierarchyList>$R$N';
MEMMOVE(ADR(arrXMLImage[nImageByte]), ADR(strString), LEN(strString));
nImageByte := nImageByte + LEN(strString);

(*****************************************************************************)


	(* update outputs *)
	bDone := TRUE;

(* unknown state *)
ELSIF bExecute = FALSE THEN

	(* clear outputs *)
	bDone := FALSE;
END_IF

END_FUNCTION_BLOCK

// ---- POUs/_Exclude/FSS2/FB_FSS2_WriteFile.TcPOU
FUNCTION_BLOCK FB_FSS2_WriteFile
VAR_INPUT
	bExecute			: BOOL;			(* scan for valid Outer in arrOuterStatus *)
	strLocalCHMPath					: STRING(255);
	strCHMFile						: T_CHM_Filename;
	nOutersPerCase						: UINT;
END_VAR
VAR_IN_OUT
	stAgregationData	 			: ST_CHM_Data;		(* case data to be written to XML *)
	stWriteCHMFileStatistic			: ST_FILE_WriteFileStatistic;
END_VAR
VAR_OUTPUT
	bDone				: BOOL;			(* TRUE = write OAC file complete *)
	bBusy				: BOOL;			(* TRUE = write OAC file in progress *)
	bError				: BOOL;			(* TRUE = write OAC file error *)
	nErrorID				: UDINT;		(* error ID *)
	nImigeProcessingSize				:UDINT;
END_VAR
VAR
	fbExecute			: R_TRIG;
	eState				: E_XML_CtrlState;
	eErrorState			: E_XML_CtrlState;

	fbBuildCHMData		: FB_FSS2_BuildXMLData;
	fbWriteFile			: FB_FILE_WriteByByte;
END_VAR

(* monitor bExecute for rising edge *)
fbExecute(CLK := bExecute);

CASE eState OF

	(* idle *)
	E_XML_IDLE:

		(* rising edge on bExecute *)
		IF fbExecute.Q = TRUE THEN

			(* update outputs *)
			bDone := FALSE;
			bBusy := TRUE;
			bError := FALSE;
			nErrorID := 0;

			eErrorState := eState;
			(* generate XML  file name and clear data for last XML file *)

			strCHMFile := F_CONCAT3('CHM_','XXXXXXXXX', '.xml');

			eState := E_XML_GENERATEIMAGE;

		(* disabled *)
		ELSIF bExecute = FALSE THEN

			(* update outputs *)
			bDone := FALSE;
			bBusy := FALSE;
			bError := FALSE;
			nErrorID := 0;
		END_IF


	(* build image in XML format *)
	E_XML_GENERATEIMAGE:

		(* build XML data *)
		fbBuildCHMData(
			bExecute		:= TRUE,
			nCartonsPerMasterCase	:=nOutersPerCase,
			stAgregationData := stAgregationData
		);

		(* build XML data complete *)
		IF fbBuildCHMData.bDone = TRUE THEN

			eState := E_XML_WRITEXML;
			nImigeProcessingSize	:= fbBuildCHMData.nImageByte;

			(* close off fbBuildXMLData *)
			fbBuildCHMData(bExecute := FALSE, stAgregationData := stAgregationData);
		END_IF


	(* write XML image *)
	E_XML_WRITEXML:

		(* write XML template to file *)
		fbWriteFile(
			bExecute	:= TRUE,
			pSourceAddr	:= ADR(fbBuildCHMData.arrXMLImage),
			nSourceSize	:= fbBuildCHMData.nImageByte,
			strPathFile	:= CONCAT(strLocalCHMPath, strCHMFile),
			tTimeout	:= T#1s
		);

		(* file write complete *)
		IF fbWriteFile.bDone = TRUE THEN

			(* file write completed OK *)
			IF fbWriteFile.bError = FALSE THEN

				;

			(* file write error *)
			ELSE

				bError := TRUE;
				nErrorID := fbWriteFile.nErrorID;
				eErrorState := eState;
			END_IF

			eState := E_XML_DONE;

			(* close of fbWriteFile *)
			fbWriteFile(bExecute := FALSE);
		END_IF


	(* XML file complete *)
	E_XML_DONE:

		(* update outputs *)
		bDone := TRUE;
		bBusy := FALSE;

		eState := E_XML_IDLE;


(* unknown state *)
ELSE

	eState := E_XML_IDLE;
END_CASE

END_FUNCTION_BLOCK

// ---- POUs/_Exclude/FSS2/FB_FSS2_WriteFileForGMES.TcPOU
FUNCTION_BLOCK FB_FSS2_WriteFileForGMES
VAR_INPUT
	bExecute			: BOOL;			(* scan for valid Outer in arrOuterStatus *)
	strLocalCHMPath					: STRING(255);
	strGMESFile						: T_CHM_Filename;
	nOutersPerCase						: UINT;
END_VAR
VAR_IN_OUT
	stAgregationData	 			: ST_CHM_Data;		(* case data to be written to XML *)
END_VAR
VAR_OUTPUT
	bDone				: BOOL;			(* TRUE = write OAC file complete *)
	bBusy				: BOOL;			(* TRUE = write OAC file in progress *)
	bError				: BOOL;			(* TRUE = write OAC file error *)
	nErrorID			: UDINT;		(* error ID *)
	nImigeProcessingSize				:UDINT;
END_VAR
VAR
	fbExecute			: R_TRIG;
	eState				: E_XML_CtrlState;
	eErrorState			: E_XML_CtrlState;

	fbBuildGMESData		: FB_FSS2_BuildXMLDataForGMES;
	fbWriteFile			: FB_FILE_WriteByByte;
END_VAR

(* monitor bExecute for rising edge *)
fbExecute(CLK := bExecute);

CASE eState OF

	(* idle *)
	E_XML_IDLE:

		(* rising edge on bExecute *)
		IF fbExecute.Q = TRUE THEN

			(* update outputs *)
			bDone := FALSE;
			bBusy := TRUE;
			bError := FALSE;
			nErrorID := 0;

			eErrorState := eState;

			(* generate XML file name and clear data for last XML file *)

			strGMESFile := F_CONCAT3('GMES_','XXXXXXXXX', '.xml');

			eState := E_XML_GENERATEIMAGE;

		(* disabled *)
		ELSIF bExecute = FALSE THEN

			(* update outputs *)
			bDone := FALSE;
			bBusy := FALSE;
			bError := FALSE;
			nErrorID := 0;
		END_IF


	(* build  image in XML format *)
	E_XML_GENERATEIMAGE:

		(* build XML data *)
		fbBuildGMESData(
			bExecute		:= TRUE,
			nCartonsPerMasterCase	:=nOutersPerCase,
			stAgregationData := stAgregationData
		);

		(* build XML data complete *)
		IF fbBuildGMESData.bDone = TRUE THEN

			eState := E_XML_WRITEXML;
			nImigeProcessingSize	:= fbBuildGMESData.nImageByte;

			(* close off fbBuildXMLData *)
			fbBuildGMESData(bExecute := FALSE, stAgregationData := stAgregationData);
		END_IF


	(* write XML image *)
	E_XML_WRITEXML:

		(* write XML template to file *)
		fbWriteFile(
			bExecute	:= TRUE,
			pSourceAddr	:= ADR(fbBuildGMESData.arrXMLImage),
			nSourceSize	:= fbBuildGMESData.nImageByte,
			strPathFile	:= CONCAT(strLocalCHMPath, strGMESFile),
			tTimeout	:= T#1s
		);

		(* file write complete *)
		IF fbWriteFile.bDone = TRUE THEN

			(* file write completed OK *)
			IF fbWriteFile.bError = FALSE THEN

				;

			(* file write error *)
			ELSE

				bError := TRUE;
				nErrorID := fbWriteFile.nErrorID;
				eErrorState := eState;
			END_IF

			eState := E_XML_DONE;

			(* close of fbWriteFile *)
			fbWriteFile(bExecute := FALSE);
		END_IF


	(* XML file complete *)
	E_XML_DONE:

		(* update outputs *)
		bDone := TRUE;
		bBusy := FALSE;

		eState := E_XML_IDLE;


(* unknown state *)
ELSE

	eState := E_XML_IDLE;
END_CASE

END_FUNCTION_BLOCK

// ---- POUs/_Exclude/FSS2/FB_FSS2_XMLImageGenerator.TcPOU
FUNCTION_BLOCK FB_FSS2_XMLImageGenerator
VAR_INPUT
	bExecute					: 	BOOL;
	strLocalCHMPath			: 	STRING(255);
	strCHMFileName			: 	T_CHM_Filename;
	strGMESFileName			: 	T_CHM_Filename;
	bCHMValideToPrint			:	BOOL;
	bClearStatistic				:	BOOL;
	nOutersPerCase			: 	UINT;
	tTimeOut					: 	TIME;
END_VAR
VAR_IN_OUT
	stCHMDataStruct			: 	ST_CHM_Data;
END_VAR
VAR_OUTPUT
	bDone					: 	BOOL;					(* TRUE = XML file write complete *)
	bBusy					: 	BOOL;					(* TRUE = XML file write in progress *)
	bError					: 	BOOL;					(* TRUE = XML file write error *)
	nErrorID					: 	UDINT;				(* file write error code *)
	stLastCaseHierarchyMessage	: 	ST_CHM_Data;
	nLastImigeSize				: 	UDINT;
	tPerformanceRate			:	TIME;

END_VAR
VAR

	nXMLStep					: 	E_XML_GeneratorState;
	eErrorState				: 	E_XML_GeneratorState;

	rtrigExecute				:	R_TRIG;
	rtrigFBDone				:	R_TRIG;

	tonTimeOut				:	TON;
	tonPerfomance			:	TON;

	fbFSS2WriteDataToXML		:	FB_FSS2_WriteFile;
	fbFSS2CreateFLGFile			:	FB_CHM_SaveFLG_File;

	fbGMESWriteDataToXML		:	FB_FSS2_WriteFileForGMES;
	fbGMESCreateFLGFile		:	FB_CHM_SaveFLG_File;

	arrImigeSize				: 	ARRAY[0..100] OF UDINT;

	bFSS2_WriteToXML			:	BOOL;
	bGMES_WriteToXML			:	BOOL;

	bFSS2_FLGFileExe			: 	BOOL;
	bGMES_FLGFileExe			:	BOOL;

	nSequenceNumber			: 	INT;

END_VAR

rtrigExecute(CLK:=bExecute);

tonTimeOut(IN:= nXMLStep<>E_XML_GENERATOR_IDLE, PT:= tTimeOut);

IF tonTimeOut.Q AND tTimeOut <> t#0ms THEN

	bDone	:=  	TRUE;
	bBusy	:=  	FALSE;
	bError	:= 	TRUE;
	nErrorID	:= 	1;

	bFSS2_WriteToXML	:=  FALSE;
	bGMES_WriteToXML	:=  FALSE;

	bFSS2_FLGFileExe	:=  FALSE;
	bGMES_FLGFileExe	:=  FALSE;

	nXMLStep	:=E_XML_GENERATOR_IDLE;
END_IF

tonPerfomance(IN:= nXMLStep<>E_XML_GENERATOR_IDLE, PT:= t#30s);

IF bClearStatistic THEN
	MEMSET(ADR(arrImigeSize), 16#00, SIZEOF(arrImigeSize));
END_IF

CASE nXMLStep OF

E_XML_GENERATOR_IDLE:

	IF rtrigExecute.Q THEN

		(* update outputs *)
		bDone := FALSE;
		bBusy := TRUE;
		bError := FALSE;
		nErrorID :=0;

		eErrorState := nXMLStep;

		bFSS2_WriteToXML	:=  FALSE;
		bGMES_WriteToXML	:=  FALSE;

		bFSS2_FLGFileExe	:=  FALSE;
		bGMES_FLGFileExe	:=  FALSE;

		nLastImigeSize		:= 0;
		tPerformanceRate		 :=t#0ms;
	
		MEMSET(ADR(stLastCaseHierarchyMessage), 16#00, SIZEOF(stLastCaseHierarchyMessage));

		nXMLStep	:=E_XML_GENERATE_BODY_CHM;

	ELSIF NOT bExecute THEN

		bDone 	:= FALSE;
		bBusy 	:= FALSE;
		bError 	:= FALSE;
		nErrorID	 := 0;

		bFSS2_WriteToXML	:=  FALSE;
		bGMES_WriteToXML	:=  FALSE;

		bFSS2_FLGFileExe	:=  FALSE;
		bGMES_FLGFileExe	:=  FALSE;

	END_IF

E_XML_GENERATE_BODY_CHM:

	bFSS2_WriteToXML := TRUE;

	IF fbFSS2WriteDataToXML.bBusy THEN

		nXMLStep	:=E_XML_DONE_BODY_CHM;
	END_IF

E_XML_DONE_BODY_CHM:

	bFSS2_WriteToXML := FALSE;

	IF	fbFSS2WriteDataToXML.bError	THEN

		bError 	:= TRUE;
		nErrorID	 := fbFSS2WriteDataToXML.nErrorID;
		eErrorState := nXMLStep;

		nXMLStep	:=E_XML_GENERATOR_DONE;

	ELSIF fbFSS2WriteDataToXML.bDone THEN

		nXMLStep	:=E_XML_GENERATE_GMES;
	END_IF

E_XML_GENERATE_GMES:

	bGMES_WriteToXML := TRUE;

	IF fbGMESWriteDataToXML.bBusy THEN
		nXMLStep	:=E_XML_DONE_GMES;
	END_IF

E_XML_DONE_GMES:

	bGMES_WriteToXML := FALSE;

	IF	fbGMESWriteDataToXML.bError	THEN

		bError 	:= TRUE;
		nErrorID	 := fbGMESWriteDataToXML.nErrorID;
		eErrorState := nXMLStep;

		nXMLStep	:=E_XML_GENERATOR_DONE;

	ELSIF fbGMESWriteDataToXML.bDone THEN

		tPerformanceRate := tonPerfomance.ET;

		IF bCHMValideToPrint THEN
			nXMLStep	:=E_XML_GENERATE_FLG;
		ELSE
			nXMLStep	:=E_XML_GENERATOR_DONE;
		END_IF
	END_IF

E_XML_GENERATE_FLG:

	bFSS2_FLGFileExe := TRUE;

	IF fbFSS2CreateFLGFile.bBusy THEN
		nXMLStep	:=E_XML_DONE_FLG;
	END_IF

E_XML_DONE_FLG:

	bFSS2_FLGFileExe := FALSE;

	IF	fbFSS2CreateFLGFile.bError	THEN

		bError 	:= TRUE;
		nErrorID	 := fbFSS2CreateFLGFile.nErrorID;
		eErrorState := nXMLStep;

		nXMLStep	:=E_XML_GENERATOR_DONE;

	ELSIF fbFSS2CreateFLGFile.bDone THEN

		nXMLStep	:=E_XML_GENERATE_GMES_FLG;
	END_IF

E_XML_GENERATE_GMES_FLG:

	bGMES_FLGFileExe := TRUE;

	IF fbGMESCreateFLGFile.bBusy THEN
		nXMLStep	:=E_XML_DONE_GMES_FLG;
	END_IF

E_XML_DONE_GMES_FLG:

	bGMES_FLGFileExe := FALSE;

	IF	fbGMESCreateFLGFile.bError	THEN

		bError 	:= TRUE;
		nErrorID	 := fbGMESCreateFLGFile.nErrorID;
		eErrorState := nXMLStep;

		nXMLStep	:=E_XML_GENERATOR_DONE;

	ELSIF fbGMESCreateFLGFile.bDone THEN

		nXMLStep	:=E_XML_GENERATOR_DONE;
	END_IF

E_XML_GENERATOR_DONE:

	nSequenceNumber	:= nSequenceNumber+1;
	MEMCPY(ADR(stLastCaseHierarchyMessage), ADR(stCHMDataStruct), SIZEOF(stCHMDataStruct));

	bDone	:=  TRUE;
	bBusy	:=  FALSE;

	nXMLStep	:=E_XML_GENERATOR_IDLE;

ELSE
	nXMLStep	:=E_XML_GENERATOR_IDLE;
END_CASE

fbFSS2WriteDataToXML(
	bExecute							:= bFSS2_WriteToXML,					(* set TRUE to write Case Produced file *)
	strLocalCHMPath					:= strLocalCHMPath,	(* path for target file C:\CaseTrace*)
	strCHMFile						:=strCHMFileName,
	nOutersPerCase					:= nOutersPerCase,
	stAgregationData					:=stCHMDataStruct,		(* case data to be written to XML *)
	stWriteCHMFileStatistic				:=stWriteCHMFileStatistic,
	bDone							=>,					(* TRUE = XML file write complete *)
	bBusy							=>,					(* TRUE = XML file write in progress *)
	bError							=> ,					(* TRUE = XML file write error *)
	nErrorID							=>,				(* file write error code *)
	nImigeProcessingSize				=>
);


rtrigFBDone(CLK:= fbFSS2WriteDataToXML.bDone);

IF	rtrigFBDone.Q	THEN
	nLastImigeSize	:= fbFSS2WriteDataToXML.nImigeProcessingSize;
	MEMMOVE(ADR(arrImigeSize[1]), ADR(arrImigeSize), SIZEOF(arrImigeSize)-SIZEOF(arrImigeSize[1]));
	arrImigeSize[0] := nLastImigeSize;
END_IF

fbGMESWriteDataToXML(
	bExecute							:= bGMES_WriteToXML,					(* set TRUE to write Case Produced file *)
	strLocalCHMPath					:= strLocalCHMPath,	(* path for target file C:\CaseTrace*)
	strGMESFile						:=strGMESFileName,
	nOutersPerCase					:= nOutersPerCase,
	stAgregationData					:=stCHMDataStruct,		(* case data to be written to XML *)
	bDone							=>,					(* TRUE = XML file write complete *)
	bBusy							=>,					(* TRUE = XML file write in progress *)
	bError							=> ,					(* TRUE = XML file write error *)
	nErrorID							=>,				(* file write error code *)
	nImigeProcessingSize				=>
);

fbFSS2CreateFLGFile(
	bExecute							:= bFSS2_FLGFileExe,					(* set TRUE to write Case Produced file *)
	sPath							:= strLocalCHMPath,			(* path for target file C:\CaseTrace*)
	sFLGFileName						:=strCHMFileName,
	bDone							=>,					(* TRUE = XML file write complete *)
	bBusy							=>,					(* TRUE = XML file write in progress *)
	bError							=>,					(* TRUE = XML file write error *)
	nErrorID							=>,				(* file write error code *)
	sFileName						=>,			(* file name generated from sCaseData *)
	nImigeProcessingSize				=>
);

fbGMESCreateFLGFile(
	bExecute							:= bGMES_FLGFileExe,					(* set TRUE to write Case Produced file *)
	sPath							:= strLocalCHMPath,			(* path for target file C:\CaseTrace*)
	sFLGFileName						:=strGMESFileName,
	bDone							=>,					(* TRUE = XML file write complete *)
	bBusy							=>,					(* TRUE = XML file write in progress *)
	bError							=>,					(* TRUE = XML file write error *)
	nErrorID							=>,				(* file write error code *)
	nImigeProcessingSize				=>
);

END_FUNCTION_BLOCK

// ---- POUs/_Exclude/F_ALARM_SetDefinition_ORG.TcPOU
(*Max text message cannot exceed 255 char including perfedeined: ('MessageTypeNo:=', INT_TO_STRING(nMessageTypeNo), ' ; MessageInfo="',sTextMessage,'"', ' ; AutoReset=', BOOL_TO_STRING(bAutoReset))*)
FUNCTION F_ALARM_SetDefinition_ORG : T_MaxString
VAR_INPUT
	bAlarmTrigger 				: BOOL;
	nCategoryNo				: INT;
	nMessageTypeNo			: INT;
	sTextMessage				: STRING(200); (* Number of 200 char + 51 char form predefined message*)
	tAlarmTimout 				: TIME :=t#1000ms;
	bAlarmDefinitionEnable 	: BOOL;
	bInhibitReset 				: BOOL;
	bInternalReset 				: BOOL;
END_VAR

VAR
	sMessagePrfix				: T_Char;
	sMessageNo				: STRING(3);

	bAutoReset 				: BOOL;
	nGroupIndex 				: INT;
	nActualAlarmPosition		: INT;
END_VAR
(*All VAR_IN_OUT variables have been moved to the end of the declaration due to compatibility reasons*)
VAR_IN_OUT
	nAlarmIndex				: INT;
	//sMSG_Info				: T_MaxString;
END_VAR

nAlarmIndex := LIMIT(0, nAlarmIndex, cMAX_MESSAGE_NUMBER);

IF nAlarmIndex <> cMAX_MESSAGE_NUMBER THEN

	IF nMessageTypeNo >= 0  AND  nMessageTypeNo <= 15 THEN

		sMessagePrfix := 'A';
		IF nMessageTypeNo > 7 THEN; 	(*Message type from 8 to 15 are set up as warrninrg*)
			bAutoReset :=TRUE;
			sMessagePrfix := 'W';
		END_IF

		sMessageNo := F_AddPadding(nAlarmIndex, 3);

		IF	 sTextMessage = '' THEN

			sTextMessage :=  F_CONCAT5('(','S',sMessageNo,') ','Missing alarm description');
			//sMSG_Info := F_CONCAT9('Cat=',INT_TO_STRING(nCategoryNo),';MsgType=', INT_TO_STRING(nMessageTypeNo),';MsgInfo="',sTextMessage,'"', ';AutoRst=', BOOL_TO_STRING(bAutoReset));
			F_ALARM_SetDefinition := F_CONCAT9('Cat=',INT_TO_STRING(nCategoryNo),';MsgType=', INT_TO_STRING(nMessageTypeNo),';MsgInfo="',sTextMessage,'"', ';AutoRst=', BOOL_TO_STRING(bAutoReset));
			//F_ALARM_SetDefinition := F_CONCAT5('MessageTypeNo:=', INT_TO_STRING(nMessageTypeNo), ' ; MessageInfo="Misssing alarm description', ' ; AutoReset=', BOOL_TO_STRING(bAutoReset));*)
		ELSE
			sTextMessage :=  F_CONCAT5('(',sMessagePrfix,sMessageNo,') ',sTextMessage);
			//sMSG_Info := F_CONCAT9('Cat=',INT_TO_STRING(nCategoryNo),';MsgType=', INT_TO_STRING(nMessageTypeNo),';MsgInfo="',sTextMessage,'"', ';AutoRst=', BOOL_TO_STRING(bAutoReset));
			F_ALARM_SetDefinition := F_CONCAT9('Cat=',INT_TO_STRING(nCategoryNo),';MsgType=', INT_TO_STRING(nMessageTypeNo),';MsgInfo="',sTextMessage,'"', ';AutoRst=', BOOL_TO_STRING(bAutoReset));
			//F_ALARM_SetDefinition := F_CONCAT7('MessageTypeNo:=', INT_TO_STRING(nMessageTypeNo), ' ; MessageInfo="',sTextMessage,'"', ' ; AutoReset=', BOOL_TO_STRING(bAutoReset));
		END_IF
	
		nGroupIndex:= nAlarmIndex/32;
		nActualAlarmPosition:= nAlarmIndex MOD 32;

		stAlarmsSettings[nGroupIndex].aTextMessageTable[nActualAlarmPosition]		:= sTextMessage;
		stAlarmsSettings[nGroupIndex].aAlarmTriggerTable[nActualAlarmPosition]		:= bAlarmTrigger ;
		(*stAlarmsSettings[nGroupIndex].aAlarmTriggerTable[nActualAlarmPosition]		:= TRUE ;*)		(*flag SET for internal force all alarms ath the same time to refresh DB*)
		stAlarmsSettings[nGroupIndex].aAlarmTimoutTable[nActualAlarmPosition]		:= tAlarmTimout;
		stAlarmsSettings[nGroupIndex].aBlockEnableTable[nActualAlarmPosition]		:= bAlarmDefinitionEnable;
		(*stAlarmsSettings[nGroupIndex].aBlockEnableTable[nActualAlarmPosition]		:= TRUE ;*)	(*flag SET for internal force all alarms ath the same time to refresh DB*)
		stAlarmsSettings[nGroupIndex].aInhibitResetTable[nActualAlarmPosition]		:= bInhibitReset AND bAlarmDefinitionEnable;
		stAlarmsSettings[nGroupIndex].aAutoResetTable[nActualAlarmPosition]			:= bAutoReset;
		stAlarmsSettings[nGroupIndex].aInternalResetTable[nActualAlarmPosition]		:= bInternalReset;
		stAlarmsSettings[nGroupIndex].aCategoryNoTable[nActualAlarmPosition]		:=nCategoryNo;
		stAlarmsSettings[nGroupIndex].aMessageTypeStatusTable[nActualAlarmPosition]	:= F_FiltredSetBitState16(TRUE, 'ALL', nMessageTypeNo, TRUE, stAlarmsSettings[nGroupIndex].aMessageTypeStatusTable[nActualAlarmPosition]);
		(*stAlarmsSettings[nGroupIndex].aMessageTypeNoTable[nActualAlarmPosition]	:=nMessageTypeNo;*)

	ELSE
		//sMSG_Info := F_CONCAT7('Cat=',INT_TO_STRING(0),';MsgType:=', INT_TO_STRING(-1),';MsgInfo="ALARM DISABLEBY BY MESSAGE TYPE', ';AutoRst=', BOOL_TO_STRING(FALSE));
		F_ALARM_SetDefinition := F_CONCAT7('Cat=',INT_TO_STRING(0),';MsgType:=', INT_TO_STRING(-1),';MsgInfo="ALARM DISABLEBY BY MESSAGE TYPE', ';AutoRst=', BOOL_TO_STRING(FALSE));
	END_IF

	nAlarmIndex := nAlarmIndex +1;
ELSE
	//sMSG_Info := F_CONCAT7('Cat=',INT_TO_STRING(0),';MsgType:=', INT_TO_STRING(-2),';MsgInfo="MESSAGE NUMBER MAX LIMIT ', ';AutoRst=', BOOL_TO_STRING(FALSE));
	F_ALARM_SetDefinition := F_CONCAT7('Cat=',INT_TO_STRING(0),';MsgType:=', INT_TO_STRING(-2),';MsgInfo="MESSAGE NUMBER MAX LIMIT ', ';AutoRst=', BOOL_TO_STRING(FALSE));

END_IF

//F_ALARM_SetDefinition := nAlarmIndex;

(*
F_ALARM_SetDefinition:= bAlarmTrigger AND bEnable;*)

END_FUNCTION

// ---- POUs/_Exclude/OAC FBs/FB_OAC_ClearArchive.TcPOU
(* scans OAC archive and deletes files and folders older than tMaxArchiveAge *)
FUNCTION_BLOCK FB_OAC_ClearArchive
VAR_INPUT
	bExecute				: BOOL;			(* set TRUE to scan archive for old folders and files *)
	strLocalOACPath		: STRING(255);	(* CaseTrace OAC folder path *)
	sSystemTime			: TIMESTRUCT;	(* current system time *)
END_VAR
VAR_OUTPUT
	bDone				: BOOL;			(* TRUE = scan complete *)
	bBusy				: BOOL;			(* TRUE = scan in progress *)
	bError				: BOOL;			(* TRUE = scan error *)
	nErrorID				: UDINT;		(* error code *)
	nFoldersDeleted		: UDINT;		(* total folders deleted *)
	nOACFilesDeleted		: UDINT;		(* total OAC files deleted *)
END_VAR
VAR
	fbExecute				: R_TRIG;
	eState				: E_OAC_State;
	eErrorState			: E_OAC_State;
	nSourceAge			: T_ULARGE_INTEGER;
	nDeleteAge			: T_ULARGE_INTEGER;
	nOACFilesFound		: UDINT;

	fbFindFile				: FB_EnumFindFileEntry;
	eFileCmd 				: E_EnumCmdType := eEnumCmd_First;
	strFileName			: STRING(255);

	fbDeleteFile			: FB_FileDelete;
	(*fbDeleteFolder			: FB_RemoveDir;*)
	sStampSystemTime		: TIMESTRUCT;
END_VAR

fbExecute(CLK := bExecute);

CASE eState OF

	(* idle *)
	E_OAC_IDLE:

		(* rising edge of bExecute *)
		IF fbExecute.Q = TRUE THEN

			(* update outputs *)
			bDone := FALSE;
			bBusy := TRUE;
			bError := FALSE;
			nErrorID := 0;

			(* reset values *)
			nOACFilesDeleted := 0;
			nOACFilesFound := 0;

			strFileName := '';
			eFileCmd := eEnumCmd_First;

			sStampSystemTime := sSystemTime;

			eState := E_OAC_FINDFILE;

		(* bExecute has been reset *)
		ELSIF bExecute = FALSE THEN

			(* reset outputs *)
			bDone := FALSE;
			bBusy := FALSE;
			bError := FALSE;
			nErrorID := 0;
		END_IF

	(* find files in folder *)
	E_OAC_FINDFILE:

		(* get list of files *)
		fbFindFile(
			sNetId		:= '',
			sPathName	:= CONCAT(strLocalOACPath, '\*.*'),
			eCmd		:= eFileCmd,
			bExecute	:= TRUE,
			tTimeout	:= T#5s
		);

		(* find date complete *)
		IF fbFindFile.bBusy = FALSE THEN

			(* find file completed OK *)
			IF fbFindFile.bError = FALSE THEN

				(* file list complete *)
				IF fbFindFile.bEOE = TRUE THEN

					eFileCmd := eEnumCmd_First;

					eState := E_OAC_IDLE;

				(* file found *)
				ELSE

					(* first 2 files could be '.' and '..' *)
					IF fbFindFile.stFindFile.sFileName = '.' OR fbFindFile.stFindFile.sFileName = '..' THEN

						(* next file *)
						eFileCmd := eEnumCmd_Next;

					(* folder found *)
					ELSE

						(* count files in folder *)
						nOACFilesFound := nOACFilesFound + 1;

						nSourceAge:= F_FileTimeToULarge(fbFindFile.stFindFile.creationTime);
						nDeleteAge:= F_FileTimeToULarge(SYSTEMTIME_TO_FILETIME(sStampSystemTime));

						IF UInt64Cmp64(nDeleteAge, nSourceAge) = 1  THEN

							(* date folder found *)
							strFileName := fbFindFile.stFindFile.sFileName;
							eState := E_OAC_DELETEFILE;

						END_IF

						(* next folder *)
						eFileCmd := eEnumCmd_Next;
					END_IF
				END_IF

			(* find file error *)
			ELSE

				(* update outputs *)
				bError := TRUE;
				nErrorID := fbFindFile.nErrID;
				eErrorState := eState;

				eFileCmd := eEnumCmd_First;

				eState := E_OAC_IDLE;
			END_IF

			(* close off fbFindFile *)
			fbFindFile(bExecute := FALSE);
		END_IF


	(* delete old file *)
	E_OAC_DELETEFILE:

		(* delete files *)
		fbDeleteFile(
			sNetId		:= '',
			sPathName	:= F_CONCAT3(strLocalOACPath, '\', strFileName),
			ePath		:= PATH_GENERIC,
			bExecute	:= TRUE,
			tTimeout	:= T#1s
		);

		(* delete file complete *)
		IF fbDeleteFile.bBusy = FALSE THEN

			(* delete file completed OK *)
			IF fbDeleteFile.bError = FALSE THEN

				(* count files deleted from current folder *)
				nOACFilesDeleted := nOACFilesDeleted + 1;
			END_IF

			eState := E_OAC_FINDFILE;

			(* close off fbDeleteFile *)
			fbDeleteFile(bExecute := FALSE);
		END_IF


	(* complete *)
	E_OAC_DONE:

		(* update outputs *)
		bBusy := FALSE;
		bDone := TRUE;

		eState := E_OAC_IDLE;


(* unknown state *)
ELSE

	eState := E_OAC_IDLE;

	bDone := FALSE;
	bBusy := FALSE;
	bError := FALSE;
	nErrorID := 0;
END_CASE

END_FUNCTION_BLOCK

// ---- POUs/_Exclude/OCV FBs/FB_OCV_ClearArchive.TcPOU
(* scans CHM archive and deletes files and folders older than tMaxArchiveAge *)
FUNCTION_BLOCK FB_OCV_ClearArchive
VAR_INPUT
	bExecute				: BOOL;			(* set TRUE to scan archive for old folders and files *)
	strLocalOCVPath		: STRING(255);	(* CaseTrace OCV folder path *)
	sSystemTime			: TIMESTRUCT;	(* current system time *)
END_VAR
VAR_OUTPUT
	bDone				: BOOL;			(* TRUE = scan complete *)
	bBusy				: BOOL;			(* TRUE = scan in progress *)
	bError				: BOOL;			(* TRUE = scan error *)
	nErrorID				: UDINT;		(* error code *)
	nFoldersDeleted		: UDINT;		(* total folders deleted *)
	nOCVFilesDeleted		: UDINT;		(* total OCV files deleted *)
END_VAR
VAR
	fbExecute				: R_TRIG;
	eState				: E_OCV_State;
	eErrorState			: E_OCV_State;
	nSourceAge			: T_ULARGE_INTEGER;
	nDeleteAge			: T_ULARGE_INTEGER;
	nOCVFilesFound		: UDINT;

	fbFindFile				: FB_EnumFindFileEntry;
	eFileCmd 				: E_EnumCmdType := eEnumCmd_First;
	strFileName			: STRING(255);
	fbDeleteFile			: FB_FileDelete;
	sStampSystemTime		: TIMESTRUCT;
END_VAR

fbExecute(CLK := bExecute);

CASE eState OF

	(* idle *)
	E_OCV_IDLE:

		(* rising edge of bExecute *)
		IF fbExecute.Q = TRUE THEN

			(* update outputs *)
			bDone := FALSE;
			bBusy := TRUE;
			bError := FALSE;
			nErrorID := 0;

			(* reset values *)
			nOCVFilesDeleted := 0;
			nOCVFilesFound := 0;

			strFileName := '';
			eFileCmd := eEnumCmd_First;

			sStampSystemTime := sSystemTime;

			eState := E_OCV_FINDFILE;

		(* bExecute has been reset *)
		ELSIF bExecute = FALSE THEN

			(* reset outputs *)
			bDone := FALSE;
			bBusy := FALSE;
			bError := FALSE;
			nErrorID := 0;
		END_IF

	(* find files in folder *)
	E_OCV_FINDFILE:

		(* get list of files *)
		fbFindFile(
			sNetId		:= '',
			sPathName	:= CONCAT(strLocalOCVPath, '\*.*'),
			eCmd		:= eFileCmd,
			bExecute	:= TRUE,
			tTimeout	:= T#5s
		);

		(* find date complete *)
		IF fbFindFile.bBusy = FALSE THEN

			(* find file completed OK *)
			IF fbFindFile.bError = FALSE THEN

				(* file list complete *)
				IF fbFindFile.bEOE = TRUE THEN

					eFileCmd := eEnumCmd_First;

					eState := E_OCV_IDLE;

				(* file found *)
				ELSE

					(* first 2 files could be '.' and '..' *)
					IF fbFindFile.stFindFile.sFileName = '.' OR fbFindFile.stFindFile.sFileName = '..' THEN

						(* next file *)
						eFileCmd := eEnumCmd_Next;

					(* folder found *)
					ELSE

						(* count files in folder *)
						nOCVFilesFound := nOCVFilesFound + 1;

						nSourceAge:= F_FileTimeToULarge(fbFindFile.stFindFile.creationTime);
						nDeleteAge:= F_FileTimeToULarge(SYSTEMTIME_TO_FILETIME(sStampSystemTime));

						IF UInt64Cmp64(nDeleteAge, nSourceAge) = 1  THEN

							(* date folder found *)
							strFileName := fbFindFile.stFindFile.sFileName;

							eState := E_OCV_DELETEFILE;

						END_IF

						(* next folder *)
						eFileCmd := eEnumCmd_Next;
					END_IF
				END_IF

			(* find file error *)
			ELSE

				(* update outputs *)
				bError := TRUE;
				nErrorID := fbFindFile.nErrID;
				eErrorState := eState;

				eFileCmd := eEnumCmd_First;

				eState := E_OCV_IDLE;
			END_IF

			(* close off fbFindFile *)
			fbFindFile(bExecute := FALSE);
		END_IF


	(* delete old file *)
	E_OCV_DELETEFILE:

		(* delete files *)
		fbDeleteFile(
			sNetId		:= '',
			sPathName	:= F_CONCAT3(strLocalOCVPath, '\', strFileName),
			ePath		:= PATH_GENERIC,
			bExecute	:= TRUE,
			tTimeout	:= T#1s
		);

		(* delete file complete *)
		IF fbDeleteFile.bBusy = FALSE THEN

			(* delete file completed OK *)
			IF fbDeleteFile.bError = FALSE THEN

				(* count files deleted from current folder *)
				nOCVFilesDeleted := nOCVFilesDeleted + 1;
			END_IF

			eState := E_OCV_FINDFILE;

			(* close off fbDeleteFile *)
			fbDeleteFile(bExecute := FALSE);
		END_IF


	(* complete *)
	E_OCV_DONE:

		(* update outputs *)
		bBusy := FALSE;
		bDone := TRUE;

		eState := E_OCV_IDLE;


(* unknown state *)
ELSE

	eState := E_OCV_IDLE;

	bDone := FALSE;
	bBusy := FALSE;
	bError := FALSE;
	nErrorID := 0;
END_CASE

END_FUNCTION_BLOCK

// ---- POUs/_Exclude/PRG_LARS_ValidationAsConfirmation_ORG.TcPOU
 PROGRAM PRG_LARS_ValidationAsConfirmation_ORG
VAR
	rtrigNewOuterArrived					: R_TRIG;
	bNewOuterIsProccesing				: BOOL;
	tonValidationTimout					: TON;
	bValidationTimeout					: BOOL;
	bValidationTimeoutReset				: BOOL;
	fbTimeoutCounter						: CTU;
	nCount									: INT;
	fbPerformance							: FB_Interval;

	fbOuterValidationCamera				: FB_SCANNER_CameraSelect;
	(*stOuterValidationCameraOptions		: ST_SCANNER_Options := (eScannerType := E_MV_420_FULL, nImageBuffer := 1, nExpectedResp := 2);*)
	fbOuterValidationEvaluation			: FB_SCANNER_Evaluation;

	fbCheckForDuplicateOuterValidation	: FB_OUTER_CheckDuplicateStatus;

	rtrigOuterValidationCameraDone		: R_TRIG;
	bOuterValidationCameraDone			: BOOL;
	bDataReadyForValidation				: BOOL;
	bQAReject								: BOOL;

	sLastImageLableString				: T_OUTER_Barcode;

	fbMoveOuterData						: FB_OUTER_MoveOuterStatus;
	fbCompleteDataFromConfirmation	: FB_OUTER_CompleteDataFromConfirmation;
	fbMETSValidateOuterForReject			: FB_OUTER_ValidateOuterForReject;
	tofValidateOuterDoneForHMI			: TOF;
	fbMasterListUpdate					: FB_OUTER_MasterListUpdate;

	stLastOuterCompleted					: ST_OUTER_Status;
	sLastReadOuterBarcode				: T_OUTER_Barcode;
	sLastReadConfPackCode1				: T_PACK_Barcode;
	nOutersCompleted						: UDINT;
	bDoneInfo								: BOOL;

	rtrigSetOuterValidationOK			: R_TRIG;
	rtrigSetOuterValidationNOK		: R_TRIG;

	rsOuterRejectStation 				: RS;
	rsOuterRejectConfirmation 		: RS;

	rtrigResetValidationStatus			: R_TRIG;

	sRejectCode						: STRING(255);
	fbArchiveInvalidOuters			: FB_OUTER_ArchiveInvalidOuters;
	aReasonForReject					: ARRAY[0..50] OF STRING(255);
	bClearList							: BOOL;

	fbOuterProduced					: FB_KPI_GenericEfficiency;
	fbOuterInspection					: FB_KPI_OutersEfficiency;

	fbOuterLevelCounter				: FB_KPI_OuterLevelCounter;

	fbQARejectCounter				: FB_CTU32;
	fbOuterValidationIndexOK			: FB_CTU32;

	ctuConsecutiveOuterRejects		: CTU;
	nActualCount						: INT;

	stDummyImageData			: ST_SCANNER_ImageData;		(* image data structure *)
	aDistanceCheck				: ARRAY[1..2] OF FB_TimeDistance;
	bResetCTU						: BOOL;
END_VAR
VAR // added by the converter: edge detectors and wires of the graphical bodies
    _w1 : BOOL;
END_VAR

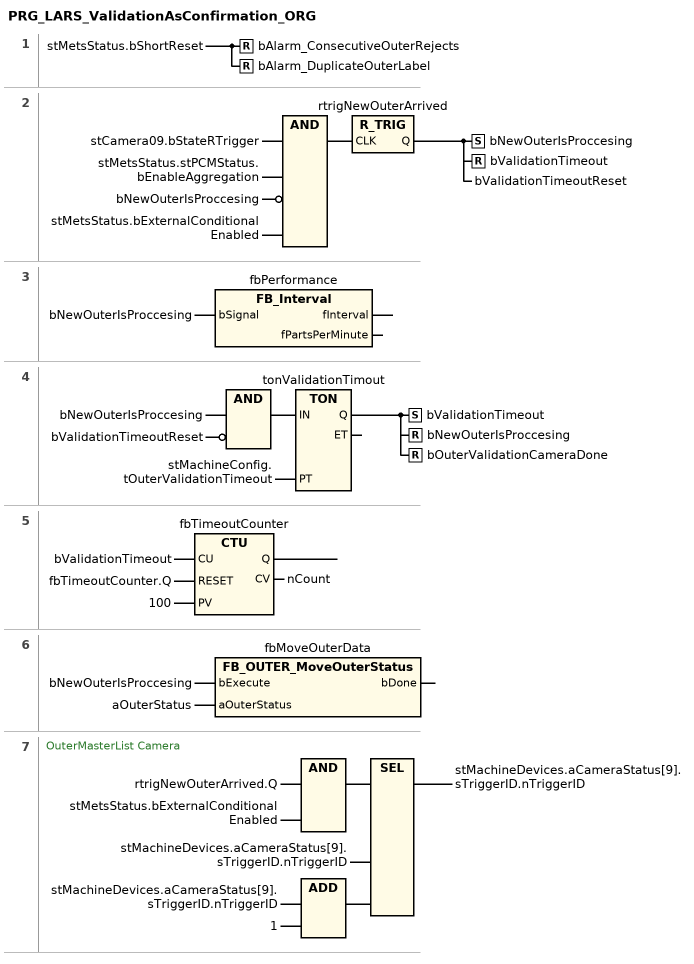
// NETWORK 1
bAlarm_ConsecutiveOuterRejects R= stMetsStatus.bShortReset;
bAlarm_DuplicateOuterLabel R= stMetsStatus.bShortReset;

// NETWORK 2
rtrigNewOuterArrived(CLK := stCamera09.bStateRTrigger AND stMetsStatus.stPCMStatus.bEnableAggregation AND NOT bNewOuterIsProccesing AND stMetsStatus.bExternalConditionalEnabled); // R_TRIG
bNewOuterIsProccesing S= rtrigNewOuterArrived.Q;
bValidationTimeout R= rtrigNewOuterArrived.Q;
bValidationTimeoutReset := rtrigNewOuterArrived.Q;

// NETWORK 3
fbPerformance(bSignal := bNewOuterIsProccesing); // FB_Interval

// NETWORK 4
tonValidationTimout(IN := bNewOuterIsProccesing AND NOT bValidationTimeoutReset, PT := stMachineConfig.tOuterValidationTimeout); // TON
bValidationTimeout S= tonValidationTimout.Q;
bNewOuterIsProccesing R= tonValidationTimout.Q;
bOuterValidationCameraDone R= tonValidationTimout.Q;

// NETWORK 5
fbTimeoutCounter(CU := bValidationTimeout, RESET := fbTimeoutCounter.Q, PV := 100, CV => nCount); // CTU

// NETWORK 6
fbMoveOuterData(bExecute := bNewOuterIsProccesing, aOuterStatus := aOuterStatus); // FB_OUTER_MoveOuterStatus

// NETWORK 7
// OuterMasterList Camera
stMachineDevices.aCameraStatus[9].sTriggerID.nTriggerID := SEL(rtrigNewOuterArrived.Q AND stMetsStatus.bExternalConditionalEnabled, stMachineDevices.aCameraStatus[9].sTriggerID.nTriggerID, stMachineDevices.aCameraStatus[9].sTriggerID.nTriggerID + 1);

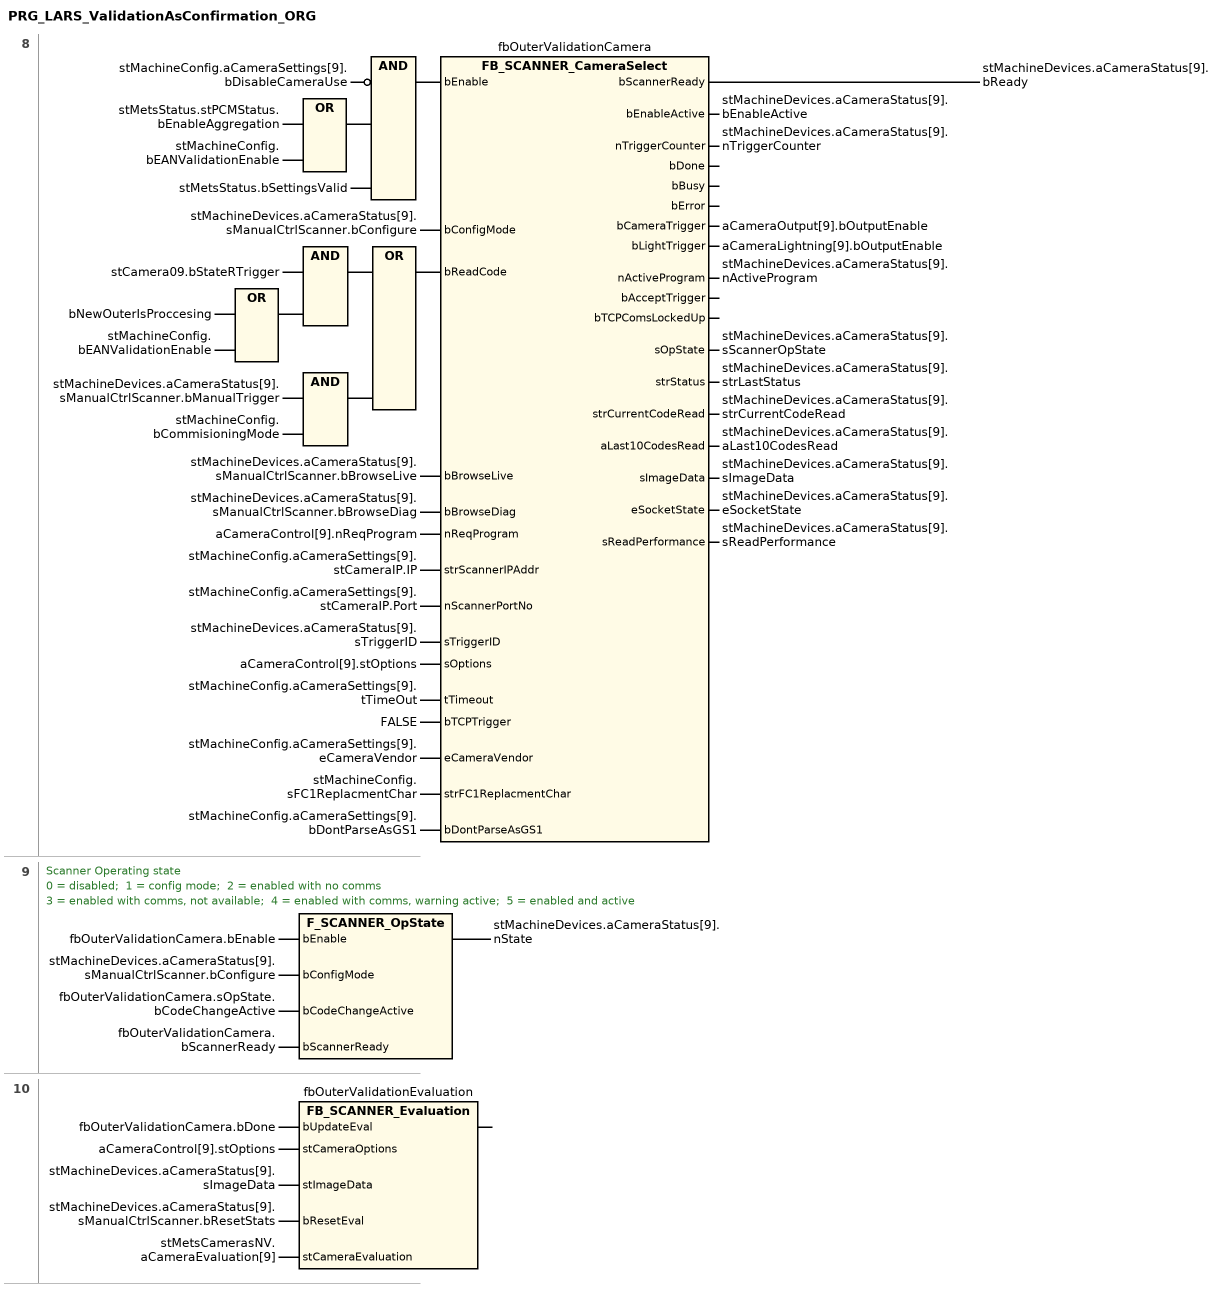
// NETWORK 8
fbOuterValidationCamera(
    bEnable := NOT stMachineConfig.aCameraSettings[9].bDisableCameraUse AND (stMetsStatus.stPCMStatus.bEnableAggregation OR stMachineConfig.bEANValidationEnable) AND stMetsStatus.bSettingsValid,
    bConfigMode := stMachineDevices.aCameraStatus[9].sManualCtrlScanner.bConfigure,
    bReadCode := stCamera09.bStateRTrigger AND (bNewOuterIsProccesing OR stMachineConfig.bEANValidationEnable) OR stMachineDevices.aCameraStatus[9].sManualCtrlScanner.bManualTrigger AND stMachineConfig.bCommisioningMode,
    bBrowseLive := stMachineDevices.aCameraStatus[9].sManualCtrlScanner.bBrowseLive,
    bBrowseDiag := stMachineDevices.aCameraStatus[9].sManualCtrlScanner.bBrowseDiag,
    nReqProgram := aCameraControl[9].nReqProgram,
    strScannerIPAddr := stMachineConfig.aCameraSettings[9].stCameraIP.IP,
    nScannerPortNo := stMachineConfig.aCameraSettings[9].stCameraIP.Port,
    sTriggerID := stMachineDevices.aCameraStatus[9].sTriggerID,
    sOptions := aCameraControl[9].stOptions,
    tTimeout := stMachineConfig.aCameraSettings[9].tTimeOut,
    bTCPTrigger := FALSE,
    eCameraVendor := stMachineConfig.aCameraSettings[9].eCameraVendor,
    strFC1ReplacmentChar := stMachineConfig.sFC1ReplacmentChar,
    bDontParseAsGS1 := stMachineConfig.aCameraSettings[9].bDontParseAsGS1,
    bEnableActive => stMachineDevices.aCameraStatus[9].bEnableActive,
    nTriggerCounter => stMachineDevices.aCameraStatus[9].nTriggerCounter,
    bCameraTrigger => aCameraOutput[9].bOutputEnable,
    bLightTrigger => aCameraLightning[9].bOutputEnable,
    nActiveProgram => stMachineDevices.aCameraStatus[9].nActiveProgram,
    sOpState => stMachineDevices.aCameraStatus[9].sScannerOpState,
    strStatus => stMachineDevices.aCameraStatus[9].strLastStatus,
    strCurrentCodeRead => stMachineDevices.aCameraStatus[9].strCurrentCodeRead,
    aLast10CodesRead => stMachineDevices.aCameraStatus[9].aLast10CodesRead,
    sImageData => stMachineDevices.aCameraStatus[9].sImageData,
    eSocketState => stMachineDevices.aCameraStatus[9].eSocketState,
    sReadPerformance => stMachineDevices.aCameraStatus[9].sReadPerformance); // FB_SCANNER_CameraSelect
stMachineDevices.aCameraStatus[9].bReady := fbOuterValidationCamera.bScannerReady;

// NETWORK 9
// 					Scanner Operating state
// 0 = disabled;  1 = config mode;  2 = enabled with no comms
// 3 = enabled with comms, not available;  4 = enabled with comms, warning active;  5 = enabled and active
//
stMachineDevices.aCameraStatus[9].nState := F_SCANNER_OpState(bEnable := fbOuterValidationCamera.bEnable, bConfigMode := stMachineDevices.aCameraStatus[9].sManualCtrlScanner.bConfigure, bCodeChangeActive := fbOuterValidationCamera.sOpState.bCodeChangeActive, bScannerReady := fbOuterValidationCamera.bScannerReady);

// NETWORK 10
fbOuterValidationEvaluation(
    bUpdateEval := fbOuterValidationCamera.bDone,
    stCameraOptions := aCameraControl[9].stOptions,
    stImageData := stMachineDevices.aCameraStatus[9].sImageData,
    bResetEval := stMachineDevices.aCameraStatus[9].sManualCtrlScanner.bResetStats,
    stCameraEvaluation := stMetsCamerasNV.aCameraEvaluation[9]); // FB_SCANNER_Evaluation

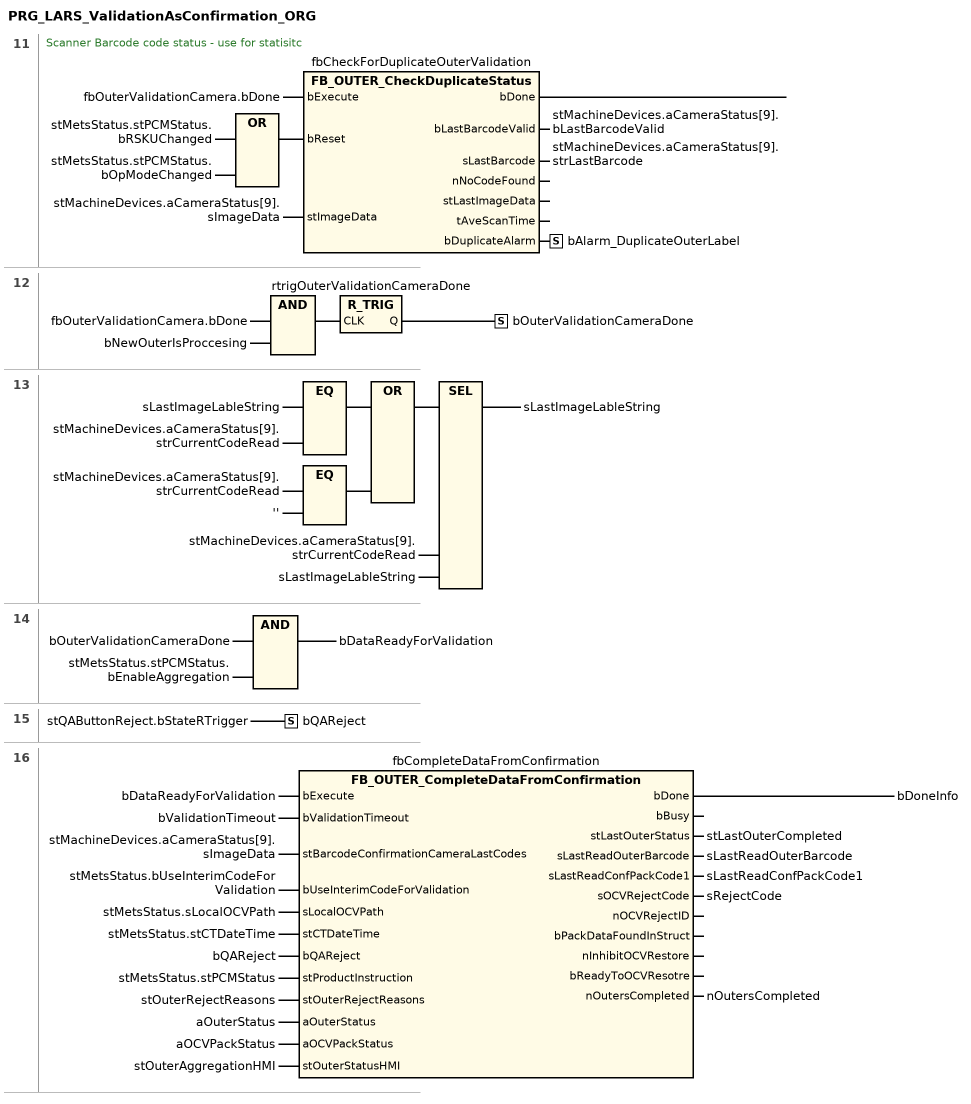
// NETWORK 11
// Scanner Barcode code status - use for statisitc
fbCheckForDuplicateOuterValidation(
    bExecute := fbOuterValidationCamera.bDone,
    bReset := stMetsStatus.stPCMStatus.bRSKUChanged OR stMetsStatus.stPCMStatus.bOpModeChanged,
    stImageData := stMachineDevices.aCameraStatus[9].sImageData,
    bLastBarcodeValid => stMachineDevices.aCameraStatus[9].bLastBarcodeValid,
    sLastBarcode => stMachineDevices.aCameraStatus[9].strLastBarcode); // FB_OUTER_CheckDuplicateStatus
bAlarm_DuplicateOuterLabel S= fbCheckForDuplicateOuterValidation.bDuplicateAlarm;

// NETWORK 12
rtrigOuterValidationCameraDone(CLK := fbOuterValidationCamera.bDone AND bNewOuterIsProccesing); // R_TRIG
bOuterValidationCameraDone S= rtrigOuterValidationCameraDone.Q;

// NETWORK 13
sLastImageLableString := SEL(sLastImageLableString = stMachineDevices.aCameraStatus[9].strCurrentCodeRead OR stMachineDevices.aCameraStatus[9].strCurrentCodeRead = '', stMachineDevices.aCameraStatus[9].strCurrentCodeRead, sLastImageLableString);

// NETWORK 14
bDataReadyForValidation := bOuterValidationCameraDone AND stMetsStatus.stPCMStatus.bEnableAggregation;

// NETWORK 15
bQAReject S= stQAButtonReject.bStateRTrigger;

// NETWORK 16
fbCompleteDataFromConfirmation(
    bExecute := bDataReadyForValidation,
    bValidationTimeout := bValidationTimeout,
    stBarcodeConfirmationCameraLastCodes := stMachineDevices.aCameraStatus[9].sImageData,
    bUseInterimCodeForValidation := stMetsStatus.bUseInterimCodeForValidation,
    sLocalOCVPath := stMetsStatus.sLocalOCVPath,
    stCTDateTime := stMetsStatus.stCTDateTime,
    bQAReject := bQAReject,
    stProductInstruction := stMetsStatus.stPCMStatus,
    stOuterRejectReasons := stOuterRejectReasons,
    aOuterStatus := aOuterStatus,
    aOCVPackStatus := aOCVPackStatus,
    stOuterStatusHMI := stOuterAggregationHMI,
    stLastOuterStatus => stLastOuterCompleted,
    sLastReadOuterBarcode => sLastReadOuterBarcode,
    sLastReadConfPackCode1 => sLastReadConfPackCode1,
    sOCVRejectCode => sRejectCode,
    nOutersCompleted => nOutersCompleted); // FB_OUTER_CompleteDataFromConfirmation
bDoneInfo := fbCompleteDataFromConfirmation.bDone;

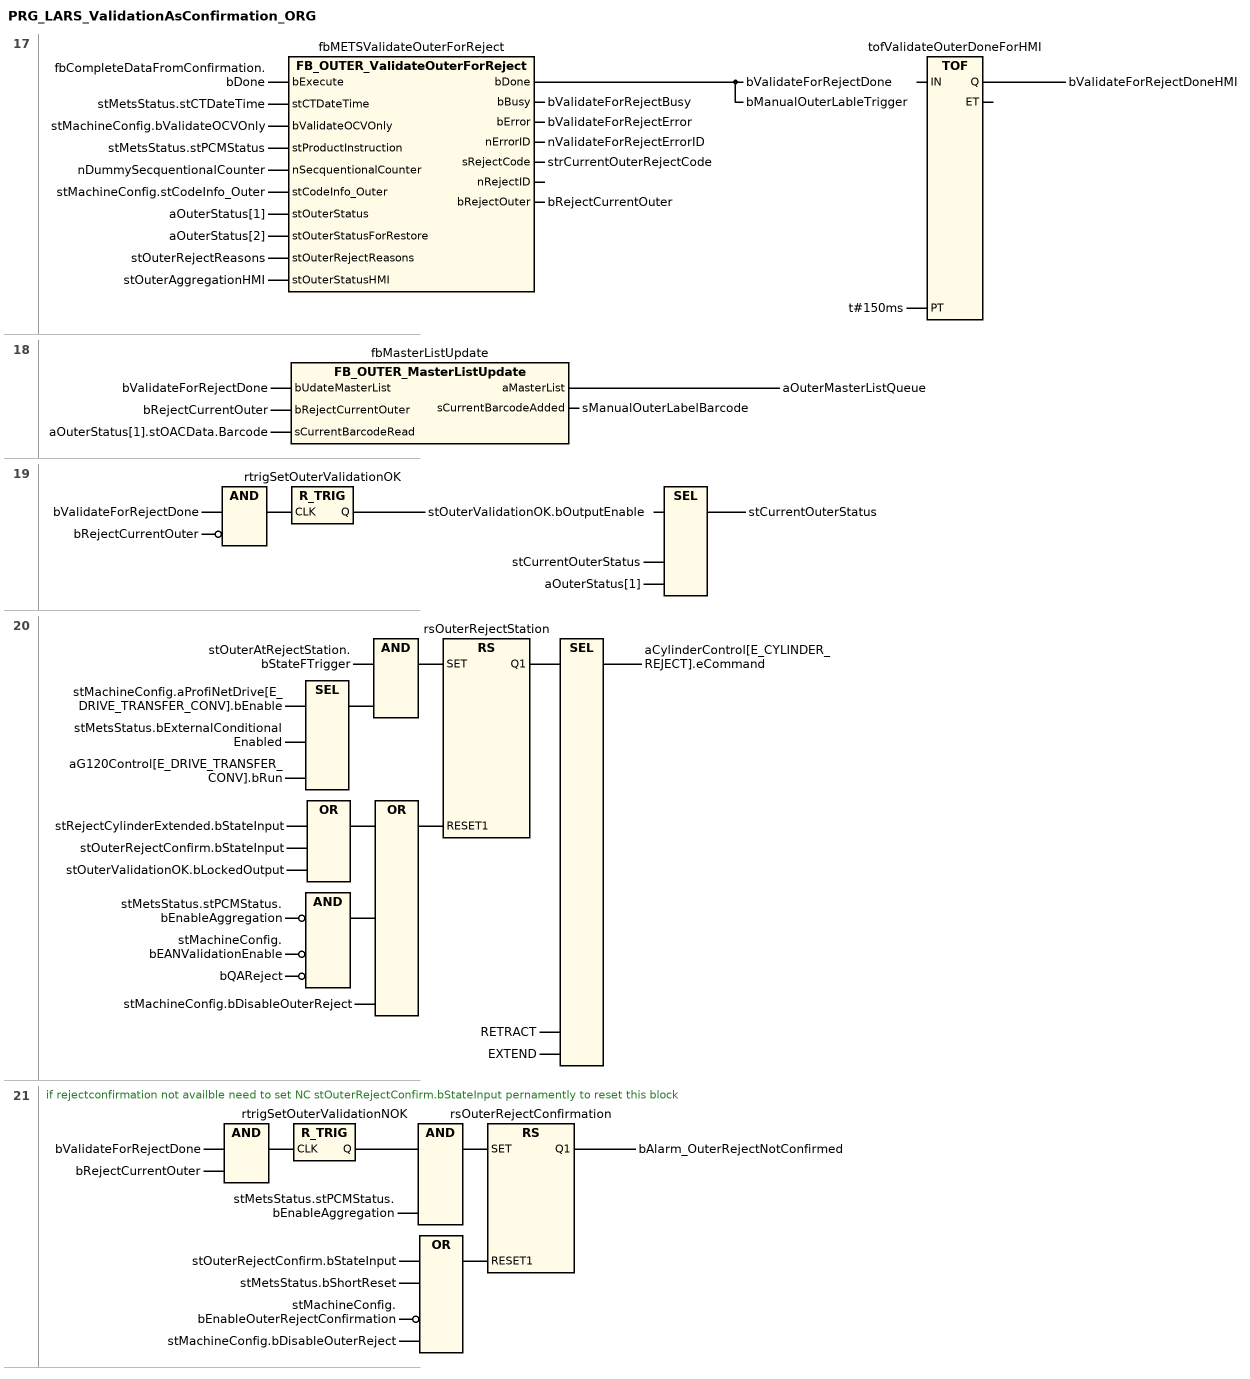
// NETWORK 17
fbMETSValidateOuterForReject(
    bExecute := fbCompleteDataFromConfirmation.bDone,
    stCTDateTime := stMetsStatus.stCTDateTime,
    bValidateOCVOnly := stMachineConfig.bValidateOCVOnly,
    stProductInstruction := stMetsStatus.stPCMStatus,
    nSecquentionalCounter := nDummySecquentionalCounter,
    stCodeInfo_Outer := stMachineConfig.stCodeInfo_Outer,
    stOuterStatus := aOuterStatus[1],
    stOuterStatusForRestore := aOuterStatus[2],
    stOuterRejectReasons := stOuterRejectReasons,
    stOuterStatusHMI := stOuterAggregationHMI,
    bBusy => bValidateForRejectBusy,
    bError => bValidateForRejectError,
    nErrorID => nValidateForRejectErrorID,
    sRejectCode => strCurrentOuterRejectCode,
    bRejectOuter => bRejectCurrentOuter); // FB_OUTER_ValidateOuterForReject
bValidateForRejectDone := fbMETSValidateOuterForReject.bDone;
bManualOuterLableTrigger := fbMETSValidateOuterForReject.bDone;
tofValidateOuterDoneForHMI(IN := fbMETSValidateOuterForReject.bDone, PT := t#150ms); // TOF
bValidateForRejectDoneHMI := tofValidateOuterDoneForHMI.Q;

// NETWORK 18
fbMasterListUpdate(
    bUdateMasterList := bValidateForRejectDone,
    bRejectCurrentOuter := bRejectCurrentOuter,
    sCurrentBarcodeRead := aOuterStatus[1].stOACData.Barcode,
    sCurrentBarcodeAdded => sManualOuterLabelBarcode); // FB_OUTER_MasterListUpdate
aOuterMasterListQueue := fbMasterListUpdate.aMasterList;

// NETWORK 19
rtrigSetOuterValidationOK(CLK := bValidateForRejectDone AND NOT bRejectCurrentOuter); // R_TRIG
stOuterValidationOK.bOutputEnable := rtrigSetOuterValidationOK.Q;
stCurrentOuterStatus := SEL(rtrigSetOuterValidationOK.Q, stCurrentOuterStatus, aOuterStatus[1]);

// NETWORK 20
rsOuterRejectStation(SET := stOuterAtRejectStation.bStateFTrigger AND SEL(stMachineConfig.aProfiNetDrive[E_DRIVE_TRANSFER_CONV].bEnable, stMetsStatus.bExternalConditionalEnabled, aG120Control[E_DRIVE_TRANSFER_CONV].bRun), RESET1 := (stRejectCylinderExtended.bStateInput OR stOuterRejectConfirm.bStateInput OR stOuterValidationOK.bLockedOutput) OR NOT stMetsStatus.stPCMStatus.bEnableAggregation AND NOT stMachineConfig.bEANValidationEnable AND NOT bQAReject OR stMachineConfig.bDisableOuterReject); // RS
aCylinderControl[E_CYLINDER_REJECT].eCommand := SEL(rsOuterRejectStation.Q1, RETRACT, EXTEND);

// NETWORK 21
// if rejectconfirmation not availble need to set NC stOuterRejectConfirm.bStateInput pernamently to reset this block
rtrigSetOuterValidationNOK(CLK := bValidateForRejectDone AND bRejectCurrentOuter); // R_TRIG
rsOuterRejectConfirmation(SET := rtrigSetOuterValidationNOK.Q AND stMetsStatus.stPCMStatus.bEnableAggregation, RESET1 := stOuterRejectConfirm.bStateInput OR stMetsStatus.bShortReset OR NOT stMachineConfig.bEnableOuterRejectConfirmation OR stMachineConfig.bDisableOuterReject); // RS
bAlarm_OuterRejectNotConfirmed := rsOuterRejectConfirmation.Q1;

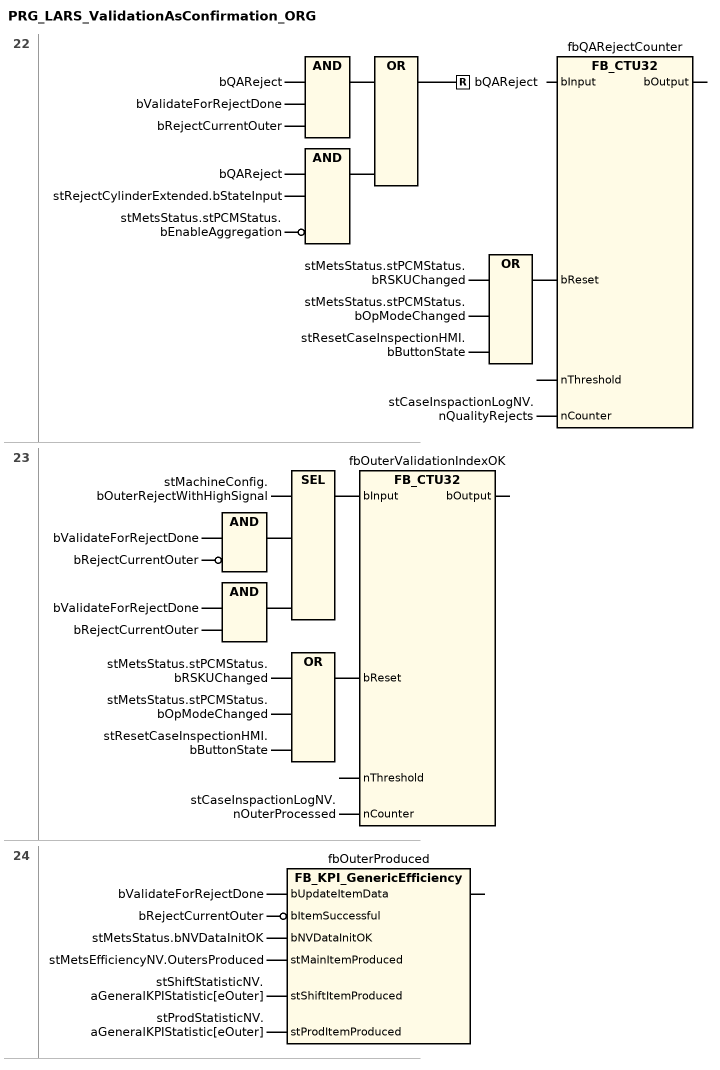
// NETWORK 22
_w1 := bQAReject AND bValidateForRejectDone AND bRejectCurrentOuter OR bQAReject AND stRejectCylinderExtended.bStateInput AND NOT stMetsStatus.stPCMStatus.bEnableAggregation;
bQAReject R= _w1;
fbQARejectCounter(
    bInput := _w1,
    bReset := stMetsStatus.stPCMStatus.bRSKUChanged OR stMetsStatus.stPCMStatus.bOpModeChanged OR stResetCaseInspectionHMI.bButtonState,
    nCounter := stCaseInspactionLogNV.nQualityRejects); // FB_CTU32

// NETWORK 23
fbOuterValidationIndexOK(
    bInput := SEL(stMachineConfig.bOuterRejectWithHighSignal, bValidateForRejectDone AND NOT bRejectCurrentOuter, bValidateForRejectDone AND bRejectCurrentOuter),
    bReset := stMetsStatus.stPCMStatus.bRSKUChanged OR stMetsStatus.stPCMStatus.bOpModeChanged OR stResetCaseInspectionHMI.bButtonState,
    nCounter := stCaseInspactionLogNV.nOuterProcessed); // FB_CTU32

// NETWORK 24
fbOuterProduced(
    bUpdateItemData := bValidateForRejectDone,
    bItemSuccessful := NOT bRejectCurrentOuter,
    bNVDataInitOK := stMetsStatus.bNVDataInitOK,
    stMainItemProduced := stMetsEfficiencyNV.OutersProduced,
    stShiftItemProduced := stShiftStatisticNV.aGeneralKPIStatistic[eOuter],
    stProdItemProduced := stProdStatisticNV.aGeneralKPIStatistic[eOuter]); // FB_KPI_GenericEfficiency

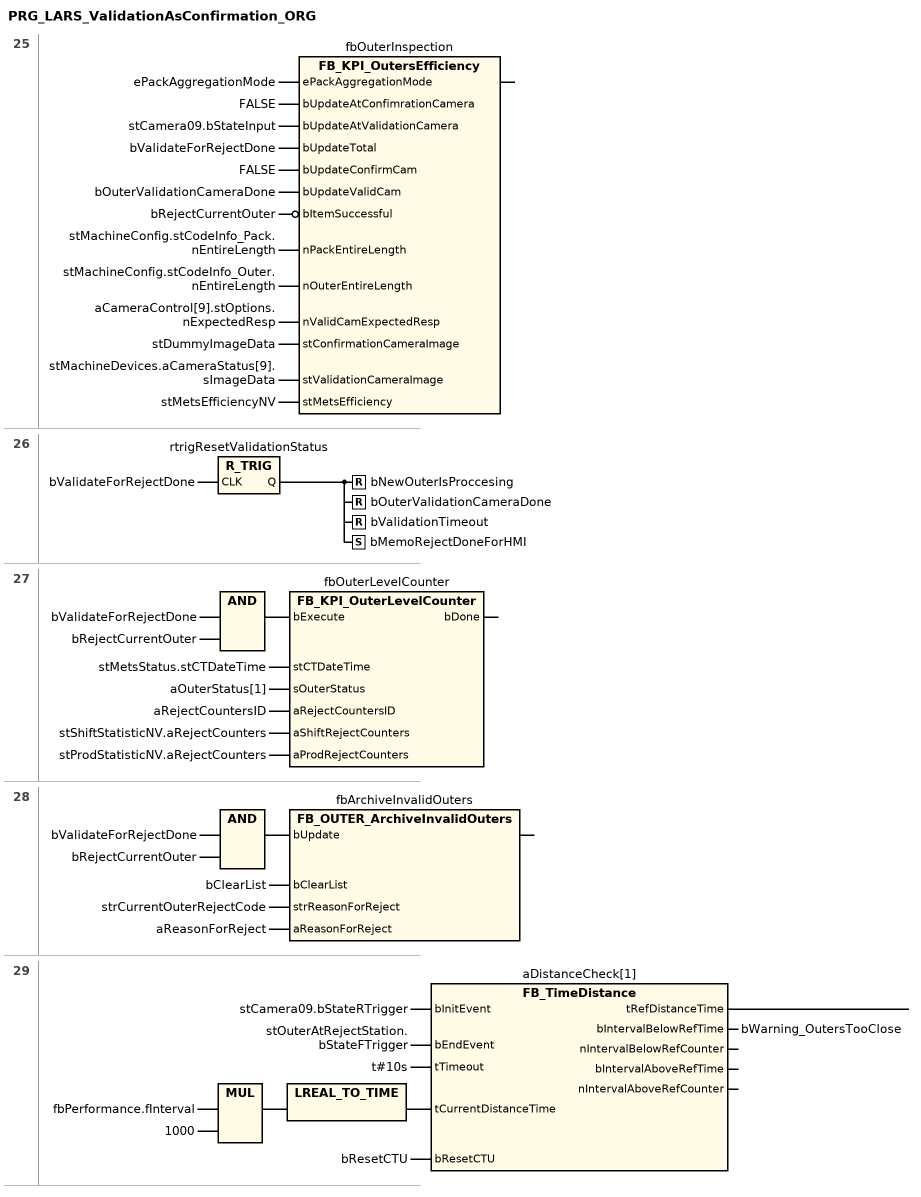
// NETWORK 25
fbOuterInspection(
    ePackAggregationMode := ePackAggregationMode,
    bUpdateAtConfimrationCamera := FALSE,
    bUpdateAtValidationCamera := stCamera09.bStateInput,
    bUpdateTotal := bValidateForRejectDone,
    bUpdateConfirmCam := FALSE,
    bUpdateValidCam := bOuterValidationCameraDone,
    bItemSuccessful := NOT bRejectCurrentOuter,
    nPackEntireLength := stMachineConfig.stCodeInfo_Pack.nEntireLength,
    nOuterEntireLength := stMachineConfig.stCodeInfo_Outer.nEntireLength,
    nValidCamExpectedResp := aCameraControl[9].stOptions.nExpectedResp,
    stConfirmationCameraImage := stDummyImageData,
    stValidationCameraImage := stMachineDevices.aCameraStatus[9].sImageData,
    stMetsEfficiency := stMetsEfficiencyNV); // FB_KPI_OutersEfficiency

// NETWORK 26
rtrigResetValidationStatus(CLK := bValidateForRejectDone); // R_TRIG
bNewOuterIsProccesing R= rtrigResetValidationStatus.Q;
bOuterValidationCameraDone R= rtrigResetValidationStatus.Q;
bValidationTimeout R= rtrigResetValidationStatus.Q;
bMemoRejectDoneForHMI S= rtrigResetValidationStatus.Q;

// NETWORK 27
fbOuterLevelCounter(
    bExecute := bValidateForRejectDone AND bRejectCurrentOuter,
    stCTDateTime := stMetsStatus.stCTDateTime,
    sOuterStatus := aOuterStatus[1],
    aRejectCountersID := aRejectCountersID,
    aShiftRejectCounters := stShiftStatisticNV.aRejectCounters,
    aProdRejectCounters := stProdStatisticNV.aRejectCounters); // FB_KPI_OuterLevelCounter

// NETWORK 28
fbArchiveInvalidOuters(
    bUpdate := bValidateForRejectDone AND bRejectCurrentOuter,
    bClearList := bClearList,
    strReasonForReject := strCurrentOuterRejectCode,
    aReasonForReject := aReasonForReject); // FB_OUTER_ArchiveInvalidOuters

// NETWORK 29
aDistanceCheck[1](
    bInitEvent := stCamera09.bStateRTrigger,
    bEndEvent := stOuterAtRejectStation.bStateFTrigger,
    tTimeout := t#10s,
    tCurrentDistanceTime := LREAL_TO_TIME(fbPerformance.fInterval * 1000),
    bResetCTU := bResetCTU,
    bIntervalBelowRefTime => bWarning_OutersTooClose); // FB_TimeDistance

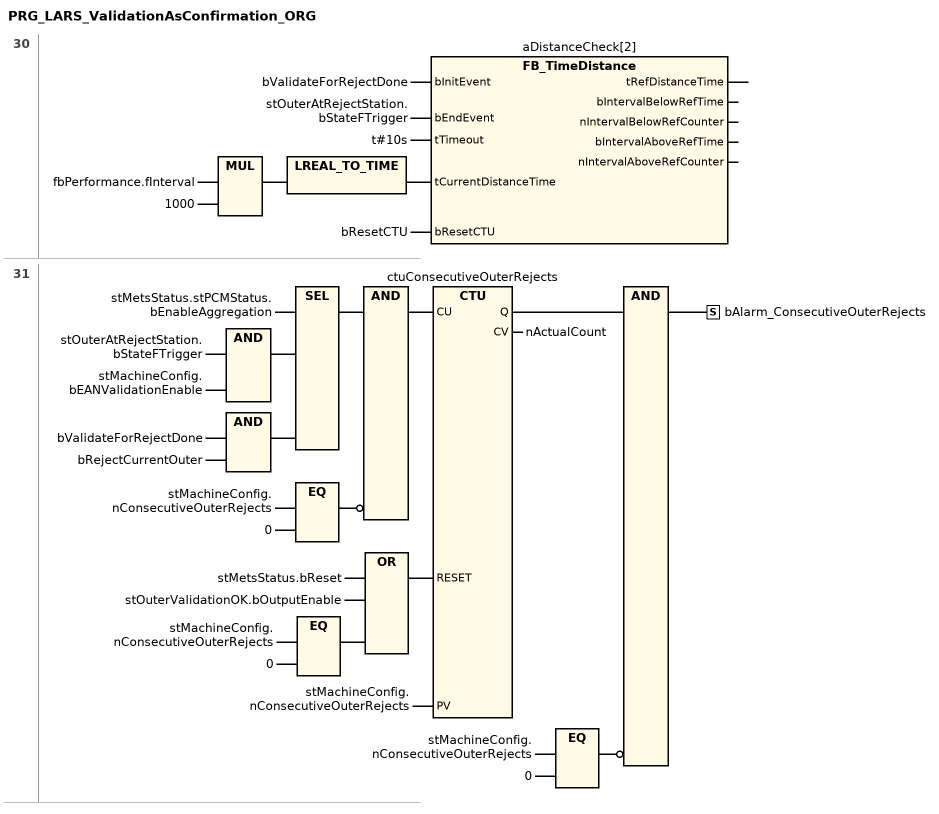
// NETWORK 30
aDistanceCheck[2](
    bInitEvent := bValidateForRejectDone,
    bEndEvent := stOuterAtRejectStation.bStateFTrigger,
    tTimeout := t#10s,
    tCurrentDistanceTime := LREAL_TO_TIME(fbPerformance.fInterval * 1000),
    bResetCTU := bResetCTU); // FB_TimeDistance

// NETWORK 31
ctuConsecutiveOuterRejects(
    CU := SEL(stMetsStatus.stPCMStatus.bEnableAggregation, stOuterAtRejectStation.bStateFTrigger AND stMachineConfig.bEANValidationEnable, bValidateForRejectDone AND bRejectCurrentOuter) AND NOT (stMachineConfig.nConsecutiveOuterRejects = 0),
    RESET := stMetsStatus.bReset OR stOuterValidationOK.bOutputEnable OR stMachineConfig.nConsecutiveOuterRejects = 0,
    PV := stMachineConfig.nConsecutiveOuterRejects,
    CV => nActualCount); // CTU
bAlarm_ConsecutiveOuterRejects S= ctuConsecutiveOuterRejects.Q AND NOT (stMachineConfig.nConsecutiveOuterRejects = 0);

END_PROGRAM

// ---- POUs/_Exclude/TestBlock_Check3.TcPOU
PROGRAM TestBlock_Check3
VAR

	sProduceDate	: STRING(14) := '20230906132030';


	sYYYY		: STRING(4);
	sMM		: STRING(2);
	sDD		: STRING(2);
	sHH		: STRING(2);
	sMMi		: STRING(2);
	sSS			: STRING(2);

	bCodeAlphaNumeric		: BOOL;
	sDateValide : BOOL;

	nCharIndex		: INT;
	sChar			: STRING(1);

END_VAR

sDateValide := TRUE;

sYYYY		:=MID(sProduceDate, 4, 1);
sMM		:=MID(sProduceDate, 2, 5);
sDD		:=MID(sProduceDate, 2, 7);
sHH		:=MID(sProduceDate, 2, 9);
sMMi		:=MID(sProduceDate, 2, 11);
sSS			:=MID(sProduceDate, 2, 13);

(* strPackCode contains data *)
IF LEN(sProduceDate) > 0 THEN

	(* check each char in the code *)
	FOR nCharIndex := 1 TO LEN(sProduceDate) DO

		(* get char from string *)
		sChar := MID(sProduceDate, 1, nCharIndex);

		(* char is every alphanumeric char *)
		IF (F_ToASC(sChar) < 16#30 OR  F_ToASC(sChar) > 16#39) THEN
			sDateValide := FALSE;
			EXIT;
		END_IF
	END_FOR
END_IF

IF sDateValide THEN

	IF STRING_TO_INT( MID(sYYYY, 2, 1)) <> 20 THEN sDateValide := FALSE; END_IF
	IF STRING_TO_INT(sMM) <1 OR  STRING_TO_INT(sMM) > 12 THEN sDateValide := FALSE; END_IF
	IF STRING_TO_INT(sDD) <1 OR  STRING_TO_INT(sDD) > 31 THEN sDateValide := FALSE; END_IF
	IF STRING_TO_INT(sHH) <0 OR  STRING_TO_INT(sHH) > 23 THEN sDateValide := FALSE; END_IF
	IF STRING_TO_INT(sMMi) <0 OR  STRING_TO_INT(sMMi) > 59 THEN sDateValide := FALSE; END_IF
	IF STRING_TO_INT(sSS) <0 OR  STRING_TO_INT(sSS) > 59 THEN sDateValide := FALSE; END_IF
END_IF

END_PROGRAM

// ---- POUs/_Exclude/TestBlock_Check4.TcPOU
 PROGRAM TestBlock_Check4
VAR

	bTest			: BOOL;
	rtTest			: R_TRIG;

	nValidatinIndex	: INT;
	nSearchIndex		: INT;

	nRemoveIndex		: INT;
	nFillUpIndex		: INT;

	stImageData				: ST_SCANNER_ImageData;
	stPackInFeedQueueTEST					: ST_PACK_InfeedQueue; (* Infeed queue *)

	bOCVStackOutOfSequence					: BOOL;

	aTESTQueue	: ARRAY[1..4] OF INT :=[ 31, 32, 33, 34];
	aPackQueue	: ARRAY[1..3] OF INT :=[ 21, 22, 23];

	bFillUp : BOOL;
	i : INT;

END_VAR

rtTest(CLK:= bTest);


IF rtTest.Q THEN

		nRemoveIndex:= 99;

		FOR nValidatinIndex := 1 TO stImageData.nCodesRead DO
			FOR nSearchIndex :=1 TO cMAX_PACK_INFEED_QUEUE DO
				IF stImageData.aCodeData[nValidatinIndex].strDataString  = stPackInFeedQueueTEST.aPackQueue[nSearchIndex].sPackCode AND
					stPackInFeedQueueTEST.aPackQueue[nSearchIndex].sPackCode <> '' THEN

					nRemoveIndex := nSearchIndex-stImageData.aCodeData[nValidatinIndex].nProgramNo;
					EXIT;
				END_IF
			END_FOR
			IF nRemoveIndex <> 99 THEN
				EXIT;
			END_IF
		END_FOR

END_IF

IF bFillUp THEN
	FOR i :=1 TO nFillUpIndex DO
		stPackInFeedQueue.aPackQueue[i].sPackCode  :=INT_TO_STRING(i);

	END_FOR
END_IF

END_PROGRAM

// ---- POUs/_Exclude/v1/FB_CAC_MoveToArchive.TcPOU
(* reads CAC files from CAC folder, deletes OAC file and copies CAC file into Archive *)
FUNCTION_BLOCK FB_CAC_MoveToArchive
VAR_INPUT
	bExecute			: BOOL;		(* set TRUE to archive OAC files *)
	strLocalOACPath		: STRING(255);	(* path to CaseTrace OAC folder *)
	strLocalCACPath		: STRING(255);	(* path to CaseTrace CAC folder *)
	strLocalOCVPath		: STRING(255);	(* path to CaseTrace OAC folder *)
	nConfirmationPack1	: INT;
	nConfirmationPack2	: INT;
	bUseInterimCodeForValidation		: BOOL;
	sSystemTime			: TIMESTRUCT;
	strPITCode				: T_CodePIT;
	strProductionOrder			: T_CodePO;
END_VAR
VAR_IN_OUT
	stCodeInfo_Pack			: ST_CodeInfo;
	stCodeInfo_Intermediate		: ST_CodeInfo;
END_VAR
VAR_OUTPUT
	bDone 				: BOOL;		(* TRUE = OAC archive complete *)
	bBusy 				: BOOL;		(* TRUE = OAC archive active *)
	bError 				: BOOL;		(* TRUE = OAC archive error *)
	nErrorID			: UDINT;	(* error code *)
	nOACFilesDeleted	: UDINT;
	nCACFilesDeleted	: UDINT;
	nOCVFilesDeleted	: UDINT;
	strCACFile			: T_CAC_Filename;
END_VAR
VAR
	fbExecute			: R_TRIG;
	eState				: E_CAC_State;
	eErrorState			: E_CAC_State;

	fbFindCACFile		: FB_EnumFindFileEntry;
	eCmdType			: E_EnumCmdType;
	fbReadCACData		: FB_XmlSrvRead;
	stCACData			: ST_CAC_Data;
	strDateFolder		: STRING(11);
	nOuterIndex			: INT;
	strOACFile			: T_OAC_Filename;
	strOCVFile			: T_OAC_Filename;
	strSerialCode			: STRING;
	aOCVFileCodeName		: ARRAY[1..2] OF T_MaxString;
	fbCreateFolder		: FB_CreateDir;
	fbDeleteFile		: FB_FileDelete;
	fbCopyFile			: FB_FILE_CopyByByte;
	(*fbMoveFile			: FB_FileRename;*)
	fbDeleteFile2			: FB_FileDelete;
END_VAR

(* monitor bExecute for rising edge *)
fbExecute(CLK := bExecute);

CASE eState OF

	(* idle *)
	E_CAC_IDLE:

		(* rising edge of bExecute *)
		IF fbExecute.Q = TRUE THEN

			(* update outputs *)
			bDone := FALSE;
			bBusy := TRUE;
			bError := FALSE;
			nErrorID := 0;
			nOACFilesDeleted := 0;
			nCACFilesDeleted := 0;
			nOCVFilesDeleted := 0;

			(* initiliase vars *)
			eCmdType := eEnumCmd_First;
			eErrorState := eState;
			MEMSET(ADR(strCACFile), 16#00, SIZEOF(strCACFile));

			eState := E_CAC_FINDFILE;

		(* bExecute has been reset *)
		ELSIF bExecute = FALSE THEN

			(* clear outputs *)
			bDone := FALSE;
			bBusy := FALSE;
			bError := FALSE;
			nErrorID := 0;
		END_IF


	(* build list of CAC files for archiving *)
	E_CAC_FINDFILE:

		(* build list *)
		fbFindCACFile(
			sNetId		:= '',
			sPathName	:= CONCAT(strLocalCACPath, 'CAC_*.xml'),
			eCmd		:= eCmdType,
			bExecute	:= TRUE,
			tTimeout	:= T#5s
		);

		(* find CAC file complete *)
		IF fbFindCACFile.bBusy = FALSE THEN

			(* find CAC file completed OK *)
			IF fbFindCACFile.bError = FALSE THEN

				(* end of CAC file list *)
				IF fbFindCACFile.bEOE = TRUE OR eCmdType = eEnumCmd_Abort THEN

					eState := E_CAC_DONE;

				(* next CAC file *)
				ELSE

					(* next CAC file *)
					strCACFile := fbFindCACFile.stFindFile.sFileName;
					eCmdType := eEnumCmd_Next;
					MEMSET(ADR(stCACData), 16#00, SIZEOF(stCACData));

					eState := E_CAC_READDATA;
				END_IF

			(* find CAC file error *)
			ELSE

				bError := TRUE;
				nErrorID := fbFindCACFile.nErrID;
				eErrorState := eState;

				eState := E_CAC_DONE;
			END_IF

			(* close off fbFindCACFile *)
			fbFindCACFile(bExecute := FALSE);
		END_IF


	(* load CAC file *)
	E_CAC_READDATA:

		(* load CAC data *)
		fbReadCACData(
			sNetId		:= '',
			ePath		:= PATH_GENERIC,
			nMode		:= XMLSRV_SKIPMISSING,
			pSymAddr	:= ADR(stCACData),
			cbSymSize	:= SIZEOF(stCACData),
			sFilePath	:= CONCAT(strLocalCACPath, strCACFile),
			sXPath		:= '/Case',
			bExecute	:= TRUE,
			tTimeout	:= T#1s
		);

		(* load CAC data complete *)
		IF fbReadCACData.bBusy = FALSE THEN

			(* load CAC data completed OK *)
			IF fbReadCACData.bError = FALSE THEN

				(* date folder as YYYYMMD\ *)
				(*strDateFolder := F_CONCAT3(F_DateCodeToDate(F_CASE_BarcodeToDateCode(stCACData.Barcode), sSystemTime), '\', '');*)
				(*strSerialCode := F_CODE_GetItem(stCACData.Barcode, eCodeAIType.SerialCode, stMAchineConfig.stCodeInfo_Case);
				strDateFolder := LEFT(strSerialCode ,7);*)
				IF strPITCode <> '' THEN
					strDateFolder := strPITCode;
				ELSIF strProductionOrder  <> '' THEN
					strDateFolder := strProductionOrder;
				ELSE
					strDateFolder := F_SYSTEM_SystemTimeToFolderName(sSystemTime);
				END_IF

				eState := E_CAC_CREATEFOLDER;

			(* load CAC data error *)
			ELSE

				bError := TRUE;
				nErrorID := fbReadCACData.nErrId;
				eErrorState := eState;

				eState := E_CAC_FINDFILE;
			END_IF

			(* close off fbReadCACData *)
			fbReadCACData(bExecute := FALSE);
		END_IF


	(* create folders *)
	E_CAC_CREATEFOLDER:

		(* create date archive folder *)
		fbCreateFolder(
			sNetId		:= '',
			sPathName	:= F_CONCAT4(strLocalCACPath, 'Archive\', strDateFolder, '\'),
			ePath		:= PATH_GENERIC,
			bExecute	:= TRUE,
			tTimeout	:= T#1s
		);

		(* create folder complete *)
		IF fbCreateFolder.bBusy = FALSE THEN

			(* create folder completed OK or folder already exists *)
			IF fbCreateFolder.bError = FALSE OR (fbCreateFolder.bError = TRUE AND fbCreateFolder.nErrId = 16#70C) THEN

				(* OAC data was active when CAC file was produced *)
				IF stCACData.CodingAndTrackingMode >= 7 THEN

					(* OAC file management required, generate OAC file name *)
					strOACFile := F_CONCAT3('OAC_', F_OUTER_BarcodeToHex(stCACData.Outer[1].Barcode), '.xml');
					(*strOACFile := F_CONCAT3('OAC_', F_SCANNER_RemoveAIBrackets(stOACData.Barcode), '.xml');*)

					nOuterIndex := 1;

					eState := E_CAC_DELETEFILE;

				(* OAC data was not active when CAC file was produced *)
				ELSE

					(* OAC file management not required*)
					eState := E_CAC_COPYFILE;
				END_IF

			(* create folder error *)
			ELSE

				(* update outputs *)
				bError := TRUE;
				nErrorID := fbCreateFolder.nErrId;
				eErrorState := eState;

				eState := E_CAC_FINDFILE;
			END_IF

			(* close off fbCreateFolder *)
			fbCreateFolder(bExecute := FALSE);
		END_IF


	(* delete OAC files *)
	E_CAC_DELETEFILE:

		(* delete OAC file *)
		fbDeleteFile(
			sNetId		:= '',
			sPathName	:= CONCAT(strLocalOACPath, strOACFile),
			ePath		:= PATH_GENERIC,
			bExecute	:= TRUE,
			tTimeout	:= T#1s
		);

		(* delete file complete *)
		IF fbDeleteFile.bBusy = FALSE THEN

			(* delete file completed OK *)
			IF fbDeleteFile.bBusy = FALSE THEN

				(* update counter *)
				nOACFilesDeleted := nOACFilesDeleted + 1;
			END_IF

			(* all OAC files archived *)
			IF nOuterIndex = stCACData.NumberOfOuters THEN

				aOCVFileCodeName[1]	:=	F_CODE_GetItem(stCACData.Outer[1].AggregationCodes[1] , eCodeAIType.SerialCode,
																	SEL(bUseInterimCodeForValidation, stCodeInfo_Pack, stCodeInfo_Intermediate));
				strOCVFile := F_CONCAT3('OCV_', F_CodeToHex(aOCVFileCodeName[1]), '.xml');
				nOuterIndex := 1;
				eState := E_CAC_DELETEOCV1;
				(*eState := E_CAC_COPYFILE;*)

			(* more OAC files to be archived *)
			ELSE

				nOuterIndex := nOuterIndex + 1;
				(* generate next OAC file name *)
				strOACFile := F_CONCAT3('OAC_', F_OUTER_BarcodeToHex(stCACData.Outer[nOuterIndex].Barcode), '.xml');
				(*strOACFile := F_CONCAT3('OAC_', F_SCANNER_RemoveAIBrackets(stOACData.Barcode), '.xml');*)

			END_IF

			(* close off fbDeleteFile *)
			fbDeleteFile(bExecute := FALSE);
		END_IF

	E_CAC_DELETEOCV1:
		(* delete 1st OCV file *)
		fbDeleteFile(
			sNetId		:= '',
			sPathName	:= CONCAT(strLocalOCVPath, strOCVFile),
			ePath		:= PATH_GENERIC,
			bExecute	:= TRUE,
			tTimeout	:= T#1s
		);

		(* delete file complete *)
		IF fbDeleteFile.bBusy = FALSE THEN

			(* delete file completed OK *)
			IF fbDeleteFile.bBusy = FALSE THEN

				(* update counter *)
				nOCVFilesDeleted := nOCVFilesDeleted + 1;
			END_IF

			(* all OAC files archived *)
			IF nOuterIndex = stCACData.NumberOfOuters THEN

				aOCVFileCodeName[2]	:=	F_CODE_GetItem(stCACData.Outer[1].AggregationCodes[2] , eCodeAIType.SerialCode,   stCodeInfo_Pack); (*no reason to have 2 diffrent intermediate codes*)
				strOCVFile := F_CONCAT3('OCV_', F_CodeToHex(aOCVFileCodeName[2]), '.xml');
				nOuterIndex := 1;
				eState := E_CAC_DELETEOCV2;

			(* more OAC files to be archived *)
			ELSE

				(* generate next OAC file name *)
				nOuterIndex := nOuterIndex + 1;
				aOCVFileCodeName[1]	:=	F_CODE_GetItem(stCACData.Outer[nOuterIndex].AggregationCodes[1] , eCodeAIType.SerialCode,
																				SEL(bUseInterimCodeForValidation, stCodeInfo_Pack, stCodeInfo_Intermediate));
				strOCVFile := F_CONCAT3('OCV_', F_CodeToHex(aOCVFileCodeName[1]), '.xml');
			END_IF

			(* close off fbDeleteFile *)
			fbDeleteFile(bExecute := FALSE);
		END_IF

	E_CAC_DELETEOCV2:
		(* delete 2nd OCV file *)
		fbDeleteFile(
			sNetId		:= '',
			sPathName	:= CONCAT(strLocalOCVPath, strOCVFile),
			ePath		:= PATH_GENERIC,
			bExecute	:= TRUE,
			tTimeout	:= T#1s
		);

		(* delete file complete *)
		IF fbDeleteFile.bBusy = FALSE THEN

			(* delete file completed OK *)
			IF fbDeleteFile.bBusy = FALSE THEN

				(* update counter *)
				nOCVFilesDeleted := nOCVFilesDeleted + 1;
			END_IF

			(* all OAC files archived *)
			IF nOuterIndex = stCACData.NumberOfOuters THEN

				eState := E_CAC_COPYFILE;

			(* more OAC files to be archived *)
			ELSE

				(* generate next OAC file name *)
				nOuterIndex := nOuterIndex + 1;
				aOCVFileCodeName[2]	:=	F_CODE_GetItem(stCACData.Outer[nOuterIndex].AggregationCodes[2] , eCodeAIType.SerialCode,   stCodeInfo_Pack);
				strOCVFile := F_CONCAT3('OCV_', F_CodeToHex(aOCVFileCodeName[2]), '.xml');
			END_IF

			(* close off fbDeleteFile *)
			fbDeleteFile(bExecute := FALSE);
		END_IF

	(* copy CAC file to archive folder *)
	E_CAC_COPYFILE:

		(* copy CAC file *)
		fbCopyFile(
			bExecute		:= TRUE,
			strPathSource	:= CONCAT(strLocalCACPath, strCACFile),
			strPathTarget	:= F_CONCAT5(strLocalCACPath, 'Archive\', strDateFolder, '\',strCACFile),
			strFileName		:= '',
			tTimeout		:= T#1s
		);

		(* copy file complete *)
		IF fbCopyFile.bBusy = FALSE THEN

			(* copy file completed OK or CAC file not found *)
			IF fbCopyFile.bError = FALSE THEN

				eState := E_CAC_MOVEFILE;

			(* copy command error *)
			ELSE

				bError := TRUE;
				nErrorID := fbCopyFile.nErrorId;
				eErrorState := eState;

				eState := E_CAC_FINDFILE;
			END_IF

			(* close off fbCopyFile *)
			fbCopyFile(bExecute := FALSE);
		END_IF


	(* delete CAC to archive folder *)
	E_CAC_MOVEFILE:

		(* delete CAC file *)
		fbDeleteFile2(
			sNetId		:= '',
			sPathName	:= CONCAT(strLocalCACPath, strCACFile),
			ePath		:= PATH_GENERIC,
			bExecute	:= TRUE,
			tTimeout	:= T#1s
		);

		(* delete file complete *)
		IF fbDeleteFile2.bBusy = FALSE THEN

			(* delete  file completed OK *)
			IF fbDeleteFile2.bError = FALSE THEN

				(* update counter *)
				nCACFilesDeleted := nCACFilesDeleted + 1;

				eState := E_CAC_FINDFILE;

			(* delete command error or file not found *)
			ELSE

				bError := TRUE;
				nErrorID := fbDeleteFile2.nErrId;
				eErrorState := eState;

				eState := E_CAC_FINDFILE;
			END_IF

			(* close off fbDeleteFile2 *)
			fbDeleteFile2(bExecute := FALSE);
		END_IF


	(* complete *)
	E_CAC_DONE:

		(* update outputs *)
		bBusy := FALSE;
		bDone := TRUE;

		eState := E_CAC_IDLE;


(* unknown state *)
ELSE

	eState := E_CAC_IDLE;
END_CASE

END_FUNCTION_BLOCK

// ---- POUs/_Exclude/v1_1/FB_CHM_BiuldXMLImige.TcPOU
FUNCTION_BLOCK FB_CHM_BiuldXMLImige
VAR_INPUT
	bExecute						: BOOL;					(* set TRUE to write Case Produced file *)
	sPath						: STRING(255);			(* path for target file C:\CaseTrace*)
	sFileName					: T_CHM_Filename;
	eMode						: E_XML_WritingMode;
	nMaxPackItem					:UINT;
	nOuterIndex					:UINT;
	bCheckFileSize					:BOOL;
	nCodingAndTrackingMode		: INT;
END_VAR
VAR_IN_OUT
	stAgregationData	 			: ST_CHM_Data;		(* case data to be written to XML *)
	stWriteCHMFileStatistic			: ST_FILE_WriteFileStatistic;
END_VAR
VAR_OUTPUT
	bDone						: BOOL;					(* TRUE = XML file write complete *)
	bBusy						: BOOL;					(* TRUE = XML file write in progress *)
	bError						: BOOL;					(* TRUE = XML file write error *)
	nErrorID						: UDINT;				(* file write error code *)
	bVerifyError					: BOOL;					(* TRUE = XML file verification error *)
	nImigeProcessingSize			:UDINT;
END_VAR
VAR
	fbExecute						: R_TRIG;
	eState						: E_XML_CtrlState;
	eErrorState					: E_XML_CtrlState;
	aXMLImage					: ARRAY[0..32767] OF BYTE;
	nImageByte					: UDINT;
	sString						: STRING(255);
	fbAppWriteFile					: FB_FILE_ApendWriteByByte;
	fbGetFileInfo					: FB_FILE_GetFileInfo;

	nPackIndex					:UINT;

	aImigeSize					: ARRAY[0..100] OF UDINT;
	nLastImigeSize					: UDINT;

END_VAR

(* rising edge of bExecute triggers new sequence *)
fbExecute(CLK := bExecute);

CASE eState OF

	(* waiting for trigger *)
	E_XML_IDLE:

		(* rising edge of bExecute *)
		IF fbExecute.Q = TRUE THEN

			(* reset internal values *)
			MEMSET(ADR(aXMLImage), 16#00, SIZEOF(aXMLImage));
			nImageByte := 0;
			eErrorState := eState;

			(* update outputs *)
			bBusy := TRUE;
			bDone := FALSE;
			bError := FALSE;
			nErrorID := 0;

			eState := E_XML_GENERATEIMAGE;

		(* bExecute has been reset *)
		ELSIF bExecute = FALSE THEN

			(* update outputs *)
			bBusy := FALSE;
			bDone := FALSE;
			bError := FALSE;
			nErrorID := 0;
			sFileName := '';
			eErrorState := E_XML_IDLE;
		END_IF


	(* generate XML image in memory *)
	E_XML_GENERATEIMAGE:

		CASE eMode OF
			E_CS_HEADER:
				A_CaseHeaderGenerator();

				nCasHeadCounter := nCasHeadCounter+1;
				nLastImigeSize	:=nImageByte;
	
				MEMMOVE(ADR(aImigeSize[1]), ADR(aImigeSize), SIZEOF(aImigeSize)-SIZEOF(aImigeSize[1]));
				aImigeSize[0] := nLastImigeSize;
	
			E_OUTER_HEADER:
				IF nCodingAndTrackingMode >= 7 THEN
					A_OuterHeaderContentGenerator();

